C03634=1032.033,-127.655,419.717,167.368,40.722,157.558
C03635=1032.027,-127.904,419.726,167.365,40.724,157.558
C03636=1032.022,-128.154,419.734,167.362,40.725,157.558
C03637=1032.017,-128.403,419.744,167.360,40.726,157.558
C03638=1032.014,-128.653,419.755,167.357,40.726,157.558
C03639=1032.010,-128.903,419.765,167.355,40.727,157.558
C03640=1032.008,-129.153,419.777,167.353,40.725,157.558
C03641=1032.006,-129.403,419.789,167.351,40.724,157.557
C03642=1032.004,-129.653,419.801,167.348,40.723,157.557
C03643=1032.004,-129.903,419.815,167.346,40.721,157.557
C03644=1032.004,-130.152,419.829,167.344,40.719,157.556
C03645=1032.005,-130.402,419.843,167.343,40.715,157.556
C03646=1032.006,-130.653,419.858,167.341,40.712,157.555
C03647=1032.008,-130.902,419.873,167.339,40.709,157.554
C03648=1032.011,-131.152,419.889,167.337,40.704,157.553
C03649=1032.014,-131.402,419.906,167.336,40.699,157.553
C03650=1032.018,-131.653,419.923,167.335,40.694,157.552
C03651=1032.023,-131.902,419.941,167.334,40.688,157.551
C03652=1032.029,-132.152,419.959,167.332,40.682,157.550
C03653=1031.703,-132.177,419.665,167.284,40.914,157.586
C03654=1031.699,-131.927,419.646,167.284,40.920,157.587
C03655=1031.694,-131.678,419.628,167.285,40.927,157.588
C03656=1031.690,-131.428,419.611,167.288,40.932,157.589
C03657=1031.686,-131.177,419.594,167.289,40.937,157.590
C03658=1031.683,-130.928,419.578,167.291,40.941,157.591
C03659=1031.681,-130.677,419.563,167.291,40.945,157.591
C03660=1031.680,-130.428,419.548,167.293,40.948,157.592
C03661=1031.679,-130.177,419.533,167.295,40.951,157.593
C03662=1031.679,-129.927,419.520,167.298,40.953,157.593
C03663=1031.680,-129.678,419.506,167.299,40.955,157.594
C03664=1031.681,-129.428,419.494,167.301,40.957,157.594
C03665=1031.683,-129.178,419.482,167.304,40.958,157.594
C03666=1031.685,-128.928,419.471,167.306,40.959,157.594
C03667=1031.689,-128.678,419.460,167.309,40.959,157.595
C03668=1031.693,-128.428,419.449,167.311,40.959,157.595
C03669=1031.696,-128.179,419.439,167.314,40.958,157.595
C03670=1031.702,-127.929,419.430,167.317,40.956,157.595
C03671=1031.708,-127.679,419.422,167.320,40.954,157.594
C03672=1031.714,-127.430,419.413,167.322,40.953,157.594
C03673=1031.719,-127.181,419.405,167.325,40.951,157.594
C03674=1031.726,-126.931,419.396,167.328,40.949,157.594
C03675=1031.731,-126.681,419.388,167.331,40.948,157.594
C03676=1031.736,-126.431,419.379,167.333,40.946,157.594
C03677=1031.743,-126.182,419.371,167.336,40.944,157.594
C03678=1031.748,-125.932,419.362,167.339,40.942,157.593
C03679=1031.755,-125.682,419.354,167.343,40.941,157.593
C03680=1031.760,-125.432,419.345,167.345,40.939,157.593
C03681=1031.766,-125.182,419.336,167.348,40.937,157.593
C03682=1031.772,-124.933,419.328,167.351,40.936,157.593
C03683=1031.778,-124.683,419.319,167.353,40.934,157.593
C03684=1031.784,-124.433,419.310,167.356,40.932,157.593
C03685=1031.790,-124.183,419.303,167.359,40.931,157.592
C03686=1031.796,-123.934,419.293,167.362,40.929,157.592
C03687=1031.801,-123.684,419.285,167.364,40.927,157.592
C03688=1031.807,-123.434,419.276,167.367,40.925,157.592
C03689=1031.813,-123.184,419.268,167.371,40.924,157.592
C03690=1031.819,-122.934,419.258,167.374,40.922,157.592
C03691=1031.824,-122.685,419.250,167.376,40.920,157.592
C03692=1031.831,-122.434,419.241,167.379,40.919,157.591
C03693=1031.837,-122.185,419.232,167.382,40.917,157.591
C03694=1031.842,-121.935,419.223,167.385,40.915,157.591
C03695=1031.848,-121.686,419.214,167.387,40.913,157.591
C03696=1031.854,-121.435,419.205,167.390,40.912,157.591
C03697=1031.860,-121.186,419.197,167.393,40.910,157.591
C03698=1031.866,-120.936,419.188,167.396,40.908,157.591
C03699=1031.871,-120.687,419.179,167.398,40.907,157.590
C03700=1031.877,-120.436,419.171,167.401,40.905,157.590
C03701=1031.883,-120.187,419.162,167.405,40.903,157.590
C03702=1031.888,-119.973,419.154,167.407,40.902,157.590
C03703=1031.893,-119.760,419.146,167.409,40.901,157.590
C03704=1031.898,-119.546,419.139,167.411,40.899,157.590
C03705=1031.903,-119.332,419.131,167.414,40.898,157.590
C03706=1031.908,-119.118,419.124,167.417,40.896,157.590
C03707=1031.914,-118.904,419.116,167.419,40.895,157.589
C03708=1031.918,-118.690,419.108,167.421,40.894,157.589
C03709=1031.924,-118.477,419.101,167.424,40.892,157.589
C03710=1031.929,-118.226,419.092,167.427,40.890,157.589
C03711=1031.936,-117.977,419.082,167.430,40.889,157.589
C03712=1031.942,-117.727,419.074,167.432,40.887,157.589
C03713=1031.948,-117.477,419.065,167.435,40.885,157.589
C03714=1031.956,-117.119,419.051,167.439,40.884,157.589
C03715=1031.965,-116.761,419.039,167.443,40.881,157.588
C03716=1031.973,-116.403,419.026,167.447,40.878,157.588
C03717=1031.981,-116.044,419.013,167.452,40.877,157.588
C03718=1031.987,-115.794,419.004,167.455,40.875,157.588
C03719=1031.994,-115.544,418.995,167.457,40.873,157.588
C03720=1031.999,-115.295,418.986,167.460,40.872,157.588
C03721=1032.005,-115.045,418.977,167.463,40.870,157.587
C03722=1032.011,-114.795,418.967,167.466,40.868,157.587
C03723=1032.016,-114.545,418.959,167.468,40.867,157.587
C03724=1032.023,-114.295,418.949,167.471,40.865,157.587
C03725=1032.029,-114.045,418.940,167.474,40.864,157.587
C03726=1032.034,-113.796,418.931,167.477,40.862,157.587
C03727=1032.040,-113.546,418.922,167.479,40.860,157.587
C03728=1032.046,-113.296,418.913,167.482,40.859,157.587
C03729=1032.052,-113.047,418.904,167.485,40.858,157.586
C03730=1032.058,-112.797,418.894,167.488,40.856,157.586
C03731=1032.064,-112.547,418.884,167.491,40.854,157.586
C03732=1032.069,-112.297,418.876,167.493,40.853,157.586
C03733=1032.075,-112.047,418.866,167.496,40.852,157.586
C03734=1032.082,-111.798,418.857,167.499,40.850,157.586
C03735=1032.087,-111.549,418.848,167.502,40.848,157.586
C03736=1032.093,-111.298,418.839,167.504,40.847,157.586
C03737=1032.099,-111.048,418.829,167.508,40.846,157.586
C03738=1032.105,-110.799,418.820,167.511,40.844,157.585
C03739=1032.111,-110.549,418.810,167.514,40.842,157.585
C03740=1032.117,-110.299,418.802,167.516,40.840,157.585
C03741=1032.123,-110.049,418.792,167.519,40.839,157.585
C03742=1032.129,-109.799,418.782,167.522,40.838,157.585
C03743=1032.135,-109.550,418.773,167.525,40.836,157.585
C03744=1032.141,-109.301,418.764,167.528,40.834,157.585
C03745=1032.147,-109.051,418.754,167.530,40.833,157.585
C03746=1032.153,-108.800,418.745,167.533,40.832,157.584
C03747=1032.159,-108.551,418.736,167.536,40.830,157.584
C03748=1032.165,-108.301,418.726,167.539,40.828,157.584
C03749=1032.171,-108.052,418.717,167.542,40.827,157.584
C03750=1032.177,-107.802,418.707,167.544,40.826,157.584
C03751=1032.183,-107.552,418.698,167.547,40.824,157.584
C03752=1032.189,-107.302,418.688,167.550,40.822,157.584
C03753=1032.195,-107.053,418.679,167.553,40.821,157.584
C03754=1032.200,-106.803,418.669,167.555,40.820,157.583
C03755=1032.206,-106.553,418.660,167.558,40.818,157.583
C03756=1032.212,-106.303,418.650,167.561,40.817,157.583
C03757=1032.219,-106.053,418.641,167.564,40.815,157.583
C03758=1032.224,-105.804,418.632,167.567,40.814,157.583
C03759=1032.230,-105.554,418.622,167.569,40.813,157.583
C03760=1032.236,-105.304,418.612,167.572,40.811,157.583
C03761=1032.242,-105.054,418.602,167.575,40.810,157.583
C03762=1032.248,-104.804,418.593,167.578,40.808,157.583
C03763=1032.254,-104.555,418.583,167.581,40.807,157.582
C03764=1032.260,-104.306,418.574,167.583,40.806,157.582
C03765=1032.265,-104.055,418.564,167.586,40.804,157.582
C03766=1032.272,-103.806,418.554,167.589,40.803,157.582
C03767=1032.278,-103.556,418.544,167.592,40.801,157.582
C03768=1032.284,-103.307,418.534,167.595,40.800,157.582
C03769=1032.290,-103.057,418.525,167.597,40.799,157.582
C03770=1032.296,-102.807,418.515,167.600,40.797,157.582
C03771=1032.302,-102.557,418.505,167.603,40.796,157.582
C03772=1032.308,-102.307,418.496,167.606,40.794,157.582
C03773=1032.314,-102.058,418.486,167.609,40.793,157.581
C03774=1032.319,-101.808,418.476,167.611,40.792,157.581
C03775=1032.325,-101.558,418.467,167.614,40.790,157.581
C03776=1032.332,-101.309,418.456,167.617,40.789,157.581
C03777=1032.338,-101.059,418.447,167.620,40.787,157.581
C03778=1032.344,-100.772,418.435,167.624,40.785,157.581
C03779=1032.351,-100.485,418.424,167.626,40.784,157.581
C03780=1032.358,-100.198,418.413,167.629,40.783,157.581
C03781=1032.365,-99.911,418.402,167.633,40.781,157.581
C03782=1032.371,-99.661,418.392,167.636,40.779,157.580
C03783=1032.377,-99.412,418.382,167.639,40.778,157.580
C03784=1032.383,-99.162,418.372,167.641,40.777,157.580
C03785=1032.389,-98.912,418.362,167.644,40.775,157.580
C03786=1032.395,-98.662,418.352,167.647,40.774,157.580
C03787=1032.401,-98.413,418.342,167.650,40.772,157.580
C03788=1032.408,-98.163,418.332,167.653,40.771,157.580
C03789=1032.414,-97.913,418.323,167.655,40.770,157.580
C03790=1032.419,-97.663,418.313,167.658,40.768,157.580
C03791=1032.426,-97.414,418.302,167.661,40.767,157.580
C03792=1032.431,-97.164,418.292,167.664,40.766,157.580
C03793=1032.437,-96.914,418.283,167.667,40.764,157.579
C03794=1032.443,-96.665,418.272,167.670,40.763,157.579
C03795=1032.449,-96.415,418.262,167.672,40.762,157.579
C03796=1032.455,-96.165,418.252,167.674,40.761,157.579
C03797=1032.461,-95.916,418.242,167.677,40.760,157.579
C03798=1032.466,-95.665,418.232,167.680,40.758,157.579
C03799=1032.473,-95.416,418.221,167.683,40.757,157.579
C03800=1032.478,-95.166,418.211,167.686,40.756,157.579
C03801=1032.485,-94.916,418.202,167.688,40.754,157.579
C03802=1032.490,-94.667,418.191,167.691,40.753,157.579
C03803=1032.496,-94.417,418.181,167.694,40.752,157.579
C03804=1032.502,-94.168,418.170,167.697,40.751,157.579
C03805=1032.508,-93.918,418.161,167.700,40.750,157.579
C03806=1032.514,-93.668,418.150,167.702,40.748,157.578
C03807=1032.520,-93.417,418.139,167.705,40.747,157.578
C03808=1032.527,-93.168,418.129,167.708,40.746,157.578
C03809=1032.532,-92.918,418.119,167.711,40.744,157.578
C03810=1032.539,-92.669,418.109,167.714,40.743,157.578
C03811=1032.544,-92.419,418.098,167.716,40.742,157.578
C03812=1032.550,-92.170,418.088,167.718,40.741,157.578
C03813=1032.556,-91.920,418.078,167.721,40.740,157.578
C03814=1032.562,-91.670,418.068,167.724,40.738,157.578
C03815=1032.568,-91.420,418.058,167.727,40.737,157.578
C03816=1032.574,-91.171,418.047,167.730,40.736,157.578
C03817=1032.580,-90.921,418.037,167.733,40.734,157.577
C03818=1032.586,-90.671,418.026,167.736,40.733,157.577
C03819=1032.593,-90.422,418.016,167.738,40.732,157.577
C03820=1032.598,-90.172,418.005,167.741,40.731,157.577
C03821=1032.604,-89.922,417.995,167.744,40.730,157.577
C03822=1032.610,-89.672,417.985,167.747,40.728,157.577
C03823=1032.616,-89.423,417.975,167.750,40.727,157.577
C03824=1032.622,-89.174,417.964,167.752,40.726,157.577
C03825=1032.628,-88.923,417.953,167.754,40.725,157.577
C03826=1032.635,-88.674,417.943,167.757,40.724,157.577
C03827=1032.640,-88.423,417.933,167.760,40.723,157.577
C03828=1032.647,-88.174,417.923,167.763,40.721,157.577
C03829=1032.652,-87.925,417.912,167.766,40.720,157.577
C03830=1032.658,-87.674,417.901,167.768,40.718,157.576
C03831=1032.665,-87.425,417.891,167.771,40.717,157.576
C03832=1032.671,-87.175,417.880,167.774,40.716,157.576
C03833=1032.677,-86.926,417.870,167.777,40.715,157.576
C03834=1032.682,-86.676,417.860,167.780,40.714,157.576
C03835=1032.689,-86.426,417.849,167.783,40.713,157.576
C03836=1032.695,-86.177,417.838,167.786,40.711,157.576
C03837=1032.701,-85.927,417.828,167.787,40.710,157.576
C03838=1032.707,-85.677,417.818,167.790,40.709,157.576
C03839=1032.713,-85.427,417.806,167.793,40.707,157.576
C03840=1032.720,-85.178,417.796,167.796,40.706,157.576
C03841=1032.725,-84.928,417.786,167.799,40.705,157.576
C03842=1032.732,-84.643,417.774,167.802,40.704,157.576
C03843=1032.740,-84.359,417.761,167.805,40.703,157.575
C03844=1032.746,-84.074,417.749,167.808,40.701,157.575
C03845=1032.753,-83.789,417.737,167.811,40.699,157.575
C03846=1032.760,-83.539,417.726,167.814,40.698,157.575
C03847=1032.766,-83.289,417.716,167.817,40.697,157.575
C03848=1032.771,-83.040,417.705,167.819,40.696,157.575
C03849=1032.779,-82.790,417.695,167.822,40.695,157.575
C03850=1032.784,-82.540,417.684,167.825,40.694,157.575
C03851=1032.790,-82.291,417.673,167.828,40.692,157.575
C03852=1032.797,-82.041,417.662,167.831,40.691,157.575
C03853=1032.803,-81.792,417.651,167.834,40.690,157.575
C03854=1032.809,-81.542,417.642,167.837,40.688,157.575
C03855=1032.815,-81.292,417.631,167.839,40.687,157.574
C03856=1032.821,-81.042,417.620,167.841,40.687,157.574
C03857=1032.828,-80.793,417.609,167.844,40.685,157.574
C03858=1032.834,-80.543,417.598,167.847,40.684,157.574
C03859=1032.840,-80.293,417.587,167.850,40.683,157.574
C03860=1032.846,-80.044,417.577,167.853,40.681,157.574
C03861=1032.852,-79.794,417.566,167.855,40.680,157.574
C03862=1032.858,-79.544,417.555,167.858,40.679,157.574
C03863=1032.864,-79.295,417.544,167.861,40.678,157.574
C03864=1032.870,-79.045,417.533,167.863,40.677,157.574
C03865=1032.876,-78.795,417.522,167.866,40.676,157.574
C03866=1032.883,-78.545,417.511,167.869,40.675,157.574
C03867=1032.889,-78.296,417.500,167.872,40.674,157.574
C03868=1032.895,-78.046,417.490,167.875,40.673,157.574
C03869=1032.901,-77.796,417.478,167.877,40.672,157.574
C03870=1032.907,-77.547,417.467,167.880,40.671,157.574
C03871=1032.912,-77.297,417.457,167.882,40.670,157.573
C03872=1032.919,-77.047,417.445,167.885,40.668,157.573
C03873=1032.924,-76.797,417.434,167.888,40.667,157.573
C03874=1032.932,-76.548,417.423,167.891,40.666,157.573
C03875=1032.938,-76.299,417.412,167.894,40.665,157.573
C03876=1032.943,-76.049,417.401,167.896,40.664,157.573
C03877=1032.950,-75.799,417.390,167.899,40.663,157.573
C03878=1032.955,-75.550,417.379,167.901,40.662,157.573
C03879=1032.962,-75.299,417.368,167.904,40.661,157.573
C03880=1032.968,-75.050,417.357,167.907,40.660,157.573
C03881=1032.974,-74.800,417.345,167.910,40.659,157.573
C03882=1032.980,-74.551,417.334,167.913,40.658,157.573
C03883=1032.986,-74.301,417.323,167.916,40.657,157.573
C03884=1032.992,-74.051,417.312,167.917,40.656,157.573
C03885=1032.998,-73.801,417.301,167.920,40.655,157.573
C03886=1033.004,-73.552,417.289,167.923,40.654,157.573
C03887=1033.010,-73.303,417.278,167.926,40.653,157.573
C03888=1033.016,-73.052,417.267,167.929,40.652,157.573
C03889=1033.022,-72.803,417.256,167.931,40.651,157.573
C03890=1033.028,-72.553,417.244,167.934,40.650,157.572
C03891=1033.034,-72.303,417.233,167.937,40.649,157.572
C03892=1033.040,-72.054,417.221,167.940,40.648,157.572
C03893=1033.046,-71.804,417.210,167.941,40.647,157.572
C03894=1033.053,-71.554,417.199,167.944,40.646,157.572
C03895=1033.058,-71.305,417.187,167.947,40.645,157.572
C03896=1033.064,-71.055,417.175,167.950,40.644,157.572
C03897=1033.070,-70.805,417.164,167.953,40.643,157.572
C03898=1033.077,-70.556,417.152,167.955,40.642,157.572
C03899=1033.082,-70.306,417.142,167.958,40.642,157.572
C03900=1033.088,-70.056,417.129,167.961,40.641,157.572
C03901=1033.094,-69.807,417.118,167.964,40.640,157.572
C03902=1033.100,-69.557,417.107,167.966,40.639,157.572
C03903=1033.106,-69.308,417.095,167.968,40.638,157.572
C03904=1033.113,-69.058,417.084,167.971,40.637,157.572
C03905=1033.118,-68.808,417.072,167.974,40.636,157.572
C03906=1033.125,-68.526,417.059,167.977,40.635,157.572
C03907=1033.132,-68.243,417.046,167.980,40.634,157.572
C03908=1033.139,-67.961,417.033,167.983,40.633,157.572
C03909=1033.146,-67.677,417.020,167.986,40.632,157.572
C03910=1033.151,-67.428,417.009,167.989,40.631,157.572
C03911=1033.158,-67.178,416.997,167.992,40.630,157.572
C03912=1033.164,-66.929,416.986,167.994,40.629,157.572
C03913=1033.170,-66.679,416.974,167.996,40.629,157.572
C03914=1033.176,-66.429,416.963,167.999,40.628,157.572
C03915=1033.182,-66.180,416.950,168.002,40.627,157.572
C03916=1033.189,-65.930,416.938,168.005,40.626,157.572
C03917=1033.194,-65.681,416.928,168.007,40.625,157.571
C03918=1033.201,-65.431,416.916,168.010,40.624,157.571
C03919=1033.206,-65.181,416.904,168.013,40.623,157.571
C03920=1033.213,-64.932,416.892,168.016,40.622,157.571
C03921=1033.219,-64.681,416.881,168.017,40.621,157.571
C03922=1033.225,-64.433,416.869,168.020,40.620,157.571
C03923=1033.231,-64.183,416.857,168.023,40.619,157.571
C03924=1033.237,-63.932,416.846,168.026,40.618,157.571
C03925=1033.243,-63.684,416.834,168.028,40.617,157.571
C03926=1033.250,-63.433,416.823,168.031,40.616,157.571
C03927=1033.256,-63.184,416.811,168.034,40.615,157.571
C03928=1033.262,-62.935,416.799,168.037,40.615,157.571
C03929=1033.268,-62.684,416.787,168.040,40.614,157.571
C03930=1033.275,-62.435,416.775,168.042,40.613,157.571
C03931=1033.281,-62.186,416.764,168.044,40.612,157.571
C03932=1033.286,-61.935,416.752,168.047,40.611,157.571
C03933=1033.293,-61.686,416.740,168.050,40.610,157.571
C03934=1033.299,-61.437,416.728,168.052,40.609,157.571
C03935=1033.305,-61.187,416.717,168.055,40.608,157.571
C03936=1033.311,-60.937,416.705,168.058,40.607,157.571
C03937=1033.318,-60.687,416.693,168.061,40.606,157.571
C03938=1033.324,-60.438,416.682,168.063,40.605,157.571
C03939=1033.330,-60.188,416.669,168.066,40.604,157.571
C03940=1033.336,-59.938,416.657,168.068,40.603,157.571
C03941=1033.343,-59.689,416.645,168.071,40.602,157.571
C03942=1033.349,-59.439,416.634,168.073,40.602,157.570
C03943=1033.354,-59.190,416.622,168.076,40.601,157.570
C03944=1033.361,-58.940,416.610,168.079,40.600,157.570
C03945=1033.368,-58.690,416.598,168.082,40.599,157.571
C03946=1033.373,-58.441,416.586,168.084,40.598,157.570
C03947=1033.379,-58.191,416.575,168.087,40.597,157.570
C03948=1033.386,-57.941,416.563,168.090,40.596,157.570
C03949=1033.393,-57.692,416.551,168.092,40.596,157.570
C03950=1033.399,-57.442,416.538,168.094,40.595,157.570
C03951=1033.405,-57.193,416.526,168.097,40.594,157.570
C03952=1033.411,-56.943,416.515,168.100,40.593,157.570
C03953=1033.417,-56.693,416.503,168.102,40.592,157.570
C03954=1033.424,-56.443,416.491,168.105,40.591,157.570
C03955=1033.430,-56.194,416.479,168.108,40.590,157.570
C03956=1033.436,-55.945,416.467,168.111,40.589,157.570
C03957=1033.442,-55.695,416.455,168.113,40.588,157.570
C03958=1033.449,-55.446,416.443,168.116,40.587,157.570
C03959=1033.455,-55.195,416.431,168.118,40.586,157.570
C03960=1033.461,-54.945,416.419,168.121,40.585,157.570
C03961=1033.468,-54.696,416.407,168.123,40.585,157.570
C03962=1033.474,-54.446,416.395,168.126,40.584,157.570
C03963=1033.480,-54.197,416.383,168.129,40.583,157.570
C03964=1033.486,-53.948,416.371,168.132,40.582,157.570
C03965=1033.493,-53.698,416.359,168.134,40.581,157.570
C03966=1033.499,-53.448,416.346,168.137,40.580,157.570
C03967=1033.505,-53.199,416.334,168.140,40.579,157.570
C03968=1033.512,-52.949,416.322,168.142,40.578,157.570
C03969=1033.519,-52.699,416.310,168.144,40.577,157.570
C03970=1033.525,-52.418,416.297,168.147,40.576,157.569
C03971=1033.533,-52.137,416.283,168.150,40.575,157.569
C03972=1033.540,-51.855,416.269,168.153,40.574,157.569
C03973=1033.547,-51.574,416.256,168.156,40.573,157.569
C03974=1033.553,-51.324,416.243,168.159,40.572,157.569
C03975=1033.560,-51.075,416.231,168.162,40.571,157.569
C03976=1033.566,-50.825,416.219,168.165,40.570,157.569
C03977=1033.572,-50.575,416.206,168.167,40.569,157.569
C03978=1033.579,-50.326,416.194,168.169,40.568,157.569
C03979=1033.585,-50.076,416.182,168.173,40.568,157.569
C03980=1033.591,-49.826,416.169,168.174,40.567,157.569
C03981=1033.597,-49.576,416.157,168.177,40.566,157.569
C03982=1033.603,-49.327,416.145,168.180,40.566,157.569
C03983=1033.609,-49.078,416.132,168.182,40.565,157.569
C03984=1033.616,-48.828,416.120,168.185,40.564,157.569
C03985=1033.621,-48.578,416.107,168.187,40.563,157.569
C03986=1033.627,-48.329,416.095,168.190,40.563,157.569
C03987=1033.634,-48.079,416.083,168.193,40.562,157.569
C03988=1033.640,-47.830,416.070,168.195,40.561,157.569
C03989=1033.646,-47.580,416.057,168.198,40.561,157.569
C03990=1033.652,-47.330,416.045,168.201,40.560,157.569
C03991=1033.659,-47.080,416.033,168.203,40.559,157.569
C03992=1033.665,-46.831,416.019,168.206,40.559,157.569
C03993=1033.671,-46.581,416.007,168.209,40.558,157.569
C03994=1033.677,-46.332,415.995,168.210,40.557,157.569
C03995=1033.683,-46.082,415.982,168.213,40.556,157.569
C03996=1033.690,-45.833,415.969,168.215,40.556,157.569
C03997=1033.696,-45.583,415.957,168.218,40.555,157.569
C03998=1033.702,-45.333,415.944,168.221,40.554,157.569
C03999=1033.708,-45.084,415.931,168.223,40.553,157.569
C04000=1033.714,-44.834,415.919,168.226,40.552,157.569
C04001=1033.721,-44.584,415.907,168.229,40.551,157.569
C04002=1033.727,-44.335,415.893,168.231,40.551,157.569
C04003=1033.733,-44.085,415.881,168.234,40.550,157.569
C04004=1033.740,-43.836,415.869,168.236,40.549,157.569
C04005=1033.746,-43.586,415.856,168.239,40.549,157.569
C04006=1033.752,-43.337,415.843,168.242,40.548,157.569
C04007=1033.758,-43.087,415.830,168.244,40.547,157.569
C04008=1033.765,-42.838,415.818,168.246,40.546,157.569
C04009=1033.771,-42.588,415.805,168.249,40.546,157.569
C04010=1033.777,-42.339,415.792,168.251,40.545,157.569
C04011=1033.783,-42.089,415.779,168.254,40.544,157.569
C04012=1033.790,-41.840,415.767,168.256,40.544,157.569
C04013=1033.796,-41.590,415.754,168.259,40.543,157.569
C04014=1033.802,-41.339,415.741,168.262,40.542,157.569
C04015=1033.808,-41.090,415.728,168.264,40.542,157.569
C04016=1033.815,-40.840,415.716,168.267,40.541,157.569
C04017=1033.821,-40.591,415.703,168.270,40.540,157.569
C04018=1033.827,-40.341,415.690,168.272,40.539,157.569
C04019=1033.833,-40.092,415.677,168.275,40.539,157.569
C04020=1033.840,-39.842,415.665,168.277,40.538,157.569
C04021=1033.846,-39.593,415.652,168.279,40.537,157.569
C04022=1033.852,-39.343,415.639,168.283,40.536,157.569
C04023=1033.859,-39.093,415.626,168.284,40.536,157.569
C04024=1033.865,-38.844,415.614,168.287,40.535,157.569
C04025=1033.872,-38.594,415.600,168.289,40.534,157.569
C04026=1033.878,-38.345,415.588,168.292,40.533,157.569
C04027=1033.884,-38.095,415.574,168.295,40.533,157.569
C04028=1033.890,-37.846,415.561,168.297,40.532,157.569
C04029=1033.896,-37.596,415.549,168.300,40.531,157.569
C04030=1033.903,-37.346,415.535,168.302,40.531,157.569
C04031=1033.909,-37.097,415.522,168.305,40.530,157.569
C04032=1033.915,-36.847,415.509,168.307,40.530,157.569
C04033=1033.921,-36.598,415.496,168.310,40.529,157.569
C04034=1033.928,-36.316,415.481,168.313,40.529,157.569
C04035=1033.935,-36.036,415.466,168.316,40.528,157.569
C04036=1033.942,-35.755,415.452,168.319,40.527,157.569
C04037=1033.948,-35.474,415.437,168.321,40.526,157.569
C04038=1033.954,-35.224,415.424,168.324,40.526,157.569
C04039=1033.961,-34.974,415.410,168.327,40.525,157.569
C04040=1033.967,-34.724,415.398,168.328,40.524,157.569
C04041=1033.973,-34.475,415.384,168.332,40.524,157.569
C04042=1033.979,-34.226,415.371,168.333,40.523,157.569
C04043=1033.986,-33.977,415.358,168.336,40.522,157.569
C04044=1033.992,-33.726,415.345,168.338,40.522,157.569
C04045=1033.998,-33.477,415.332,168.341,40.521,157.569
C04046=1034.005,-33.228,415.318,168.343,40.521,157.569
C04047=1034.011,-32.978,415.305,168.346,40.520,157.569
C04048=1034.017,-32.728,415.292,168.348,40.520,157.569
C04049=1034.024,-32.478,415.279,168.351,40.519,157.569
C04050=1034.030,-32.229,415.266,168.354,40.518,157.569
C04051=1034.036,-31.980,415.252,168.356,40.517,157.569
C04052=1034.043,-31.730,415.239,168.359,40.516,157.569
C04053=1034.049,-31.480,415.226,168.361,40.516,157.569
C04054=1034.055,-31.231,415.213,168.364,40.515,157.569
C04055=1034.061,-30.982,415.200,168.366,40.515,157.569
C04056=1034.068,-30.732,415.186,168.369,40.514,157.569
C04057=1034.074,-30.482,415.173,168.371,40.514,157.569
C04058=1034.080,-30.233,415.159,168.374,40.513,157.569
C04059=1034.087,-29.984,415.146,168.375,40.512,157.569
C04060=1034.093,-29.733,415.133,168.379,40.512,157.569
C04061=1034.099,-29.484,415.120,168.380,40.511,157.569
C04062=1034.106,-29.235,415.107,168.383,40.511,157.569
C04063=1034.112,-28.985,415.093,168.386,40.510,157.569
C04064=1034.119,-28.735,415.080,168.388,40.509,157.569
C04065=1034.125,-28.486,415.067,168.391,40.508,157.569
C04066=1034.131,-28.236,415.052,168.393,40.508,157.569
C04067=1034.137,-27.987,415.039,168.396,40.507,157.569
C04068=1034.143,-27.737,415.026,168.398,40.506,157.569
C04069=1034.150,-27.487,415.012,168.401,40.506,157.569
C04070=1034.156,-27.238,414.999,168.403,40.505,157.569
C04071=1034.163,-26.989,414.986,168.406,40.505,157.569
C04072=1034.169,-26.739,414.972,168.408,40.504,157.569
C04073=1034.175,-26.489,414.958,168.411,40.504,157.569
C04074=1034.181,-26.240,414.945,168.413,40.503,157.569
C04075=1034.188,-25.990,414.931,168.416,40.503,157.569
C04076=1034.193,-25.741,414.917,168.418,40.502,157.569
C04077=1034.200,-25.491,414.904,168.421,40.501,157.569
C04078=1034.206,-25.241,414.890,168.423,40.501,157.569
C04079=1034.213,-24.992,414.877,168.426,40.500,157.569
C04080=1034.218,-24.742,414.863,168.428,40.500,157.569
C04081=1034.225,-24.492,414.850,168.431,40.499,157.569
C04082=1034.231,-24.243,414.836,168.433,40.499,157.569
C04083=1034.237,-23.993,414.822,168.435,40.499,157.569
C04084=1034.243,-23.744,414.809,168.437,40.498,157.569
C04085=1034.250,-23.495,414.795,168.440,40.497,157.569
C04086=1034.256,-23.245,414.781,168.442,40.497,157.569
C04087=1034.262,-22.995,414.767,168.444,40.496,157.569
C04088=1034.268,-22.746,414.754,168.447,40.496,157.569
C04089=1034.274,-22.496,414.740,168.449,40.495,157.569
C04090=1034.281,-22.247,414.727,168.452,40.495,157.569
C04091=1034.288,-21.997,414.712,168.454,40.494,157.569
C04092=1034.293,-21.748,414.698,168.457,40.494,157.569
C04093=1034.300,-21.499,414.685,168.459,40.493,157.569
C04094=1034.306,-21.249,414.671,168.462,40.492,157.569
C04095=1034.312,-20.999,414.658,168.464,40.492,157.569
C04096=1034.319,-20.750,414.643,168.467,40.491,157.569
C04097=1034.325,-20.500,414.630,168.469,40.491,157.569
C04098=1034.332,-20.218,414.615,168.472,40.490,157.569
C04099=1034.339,-19.937,414.599,168.475,40.490,157.569
C04100=1034.347,-19.654,414.583,168.477,40.489,157.569
C04101=1034.353,-19.373,414.568,168.480,40.489,157.569
C04102=1034.360,-19.123,414.554,168.483,40.488,157.569
C04103=1034.366,-18.874,414.540,168.485,40.487,157.569
C04104=1034.373,-18.624,414.526,168.487,40.487,157.569
C04105=1034.378,-18.375,414.512,168.490,40.486,157.569
C04106=1034.385,-18.125,414.498,168.492,40.485,157.569
C04107=1034.392,-17.876,414.484,168.495,40.485,157.569
C04108=1034.398,-17.626,414.470,168.497,40.485,157.569
C04109=1034.404,-17.377,414.457,168.500,40.484,157.569
C04110=1034.411,-17.127,414.443,168.502,40.484,157.569
C04111=1034.417,-16.878,414.429,168.505,40.483,157.569
C04112=1034.423,-16.628,414.415,168.507,40.483,157.569
C04113=1034.429,-16.379,414.400,168.509,40.482,157.569
C04114=1034.436,-16.129,414.387,168.511,40.481,157.569
C04115=1034.442,-15.880,414.373,168.513,40.481,157.569
C04116=1034.449,-15.630,414.359,168.516,40.480,157.569
C04117=1034.455,-15.380,414.345,168.518,40.479,157.569
C04118=1034.461,-15.131,414.330,168.521,40.479,157.569
C04119=1034.468,-14.881,414.317,168.523,40.479,157.569
C04120=1034.474,-14.632,414.302,168.525,40.479,157.569
C04121=1034.481,-14.382,414.289,168.528,40.478,157.569
C04122=1034.486,-14.133,414.274,168.530,40.477,157.569
C04123=1034.492,-13.883,414.260,168.533,40.477,157.569
C04124=1034.499,-13.634,414.246,168.535,40.476,157.569
C04125=1034.505,-13.384,414.232,168.537,40.476,157.569
C04126=1034.511,-13.135,414.217,168.540,40.476,157.569
C04127=1034.518,-12.885,414.203,168.542,40.475,157.569
C04128=1034.523,-12.636,414.189,168.545,40.475,157.570
C04129=1034.530,-12.386,414.175,168.547,40.474,157.570
C04130=1034.537,-12.136,414.160,168.549,40.474,157.569
C04131=1034.542,-11.887,414.146,168.552,40.473,157.570
C04132=1034.549,-11.638,414.132,168.554,40.473,157.570
C04133=1034.555,-11.389,414.117,168.557,40.473,157.570
C04134=1034.562,-11.139,414.104,168.559,40.472,157.570
C04135=1034.568,-10.890,414.089,168.561,40.472,157.570
C04136=1034.574,-10.639,414.075,168.564,40.471,157.570
C04137=1034.581,-10.390,414.061,168.566,40.470,157.570
C04138=1034.587,-10.141,414.046,168.569,40.470,157.570
C04139=1034.593,-9.891,414.032,168.571,40.470,157.570
C04140=1034.600,-9.641,414.017,168.573,40.469,157.570
C04141=1034.605,-9.392,414.004,168.576,40.469,157.570
C04142=1034.612,-9.142,413.989,168.578,40.469,157.570
C04143=1034.618,-8.894,413.975,168.580,40.468,157.570
C04144=1034.624,-8.643,413.960,168.583,40.467,157.570
C04145=1034.631,-8.394,413.945,168.585,40.467,157.570
C04146=1034.637,-8.145,413.931,168.588,40.466,157.570
C04147=1034.643,-7.895,413.917,168.590,40.466,157.570
C04148=1034.650,-7.645,413.903,168.592,40.466,157.570
C04149=1034.656,-7.396,413.888,168.595,40.465,157.570
C04150=1034.662,-7.146,413.874,168.597,40.465,157.570
C04151=1034.669,-6.897,413.860,168.599,40.464,157.570
C04152=1034.675,-6.648,413.845,168.602,40.464,157.570
C04153=1034.681,-6.398,413.830,168.604,40.463,157.570
C04154=1034.688,-6.148,413.817,168.607,40.463,157.570
C04155=1034.695,-5.899,413.802,168.609,40.462,157.570
C04156=1034.700,-5.650,413.787,168.611,40.462,157.570
C04157=1034.708,-5.400,413.773,168.614,40.461,157.570
C04158=1034.714,-5.150,413.758,168.616,40.461,157.570
C04159=1034.719,-4.901,413.744,168.618,40.461,157.570
C04160=1034.727,-4.652,413.729,168.620,40.460,157.570
C04161=1034.733,-4.402,413.715,168.622,40.459,157.570
C04162=1034.740,-4.119,413.698,168.626,40.459,157.570
C04163=1034.747,-3.835,413.682,168.628,40.458,157.570
C04164=1034.754,-3.552,413.665,168.630,40.458,157.570
C04165=1034.762,-3.269,413.648,168.633,40.458,157.570
C04166=1034.768,-3.019,413.633,168.635,40.457,157.570
C04167=1034.774,-2.769,413.619,168.639,40.457,157.571
C04168=1034.780,-2.520,413.605,168.640,40.456,157.570
C04169=1034.786,-2.270,413.590,168.642,40.456,157.571
C04170=1034.793,-2.021,413.575,168.644,40.456,157.571
C04171=1034.798,-1.772,413.560,168.647,40.456,157.571
C04172=1034.805,-1.522,413.545,168.650,40.455,157.571
C04173=1034.811,-1.272,413.530,168.652,40.455,157.571
C04174=1034.817,-1.023,413.515,168.654,40.454,157.571
C04175=1034.823,-0.774,413.501,168.656,40.454,157.571
C04176=1034.830,-0.524,413.486,168.658,40.454,157.571
C04177=1034.836,-0.274,413.471,168.662,40.453,157.571
C04178=1034.842,-0.025,413.456,168.664,40.453,157.571
C04179=1034.848,0.224,413.441,168.666,40.453,157.571
C04180=1034.855,0.474,413.426,168.667,40.452,157.571
C04181=1034.861,0.724,413.411,168.670,40.452,157.571
C04182=1034.867,0.973,413.397,168.672,40.452,157.571
C04183=1034.873,1.222,413.382,168.675,40.451,157.571
C04184=1034.880,1.472,413.367,168.678,40.451,157.571
C04185=1034.886,1.722,413.352,168.680,40.451,157.571
C04186=1034.892,1.971,413.337,168.681,40.450,157.571
C04187=1034.899,2.220,413.321,168.684,40.450,157.571
C04188=1034.905,2.469,413.307,168.687,40.450,157.571
C04189=1034.911,2.719,413.292,168.689,40.449,157.571
C04190=1034.918,2.968,413.277,168.691,40.449,157.571
C04191=1034.924,3.218,413.262,168.693,40.448,157.571
C04192=1034.930,3.468,413.247,168.695,40.448,157.571
C04193=1034.936,3.717,413.232,168.697,40.448,157.571
C04194=1034.942,3.966,413.218,168.701,40.447,157.572
C04195=1034.948,4.216,413.202,168.703,40.447,157.572
C04196=1034.955,4.465,413.186,168.704,40.446,157.572
C04197=1034.961,4.715,413.171,168.706,40.446,157.572
C04198=1034.968,4.965,413.156,168.709,40.446,157.572
C04199=1034.973,5.214,413.142,168.712,40.446,157.572
C04200=1034.980,5.463,413.127,168.714,40.446,157.572
C04201=1034.986,5.713,413.112,168.716,40.445,157.572
C04202=1034.993,5.962,413.096,168.718,40.444,157.572
C04203=1034.999,6.212,413.081,168.720,40.444,157.572
C04204=1035.006,6.461,413.066,168.723,40.444,157.572
C04205=1035.012,6.711,413.051,168.726,40.444,157.572
C04206=1035.018,6.961,413.037,168.727,40.443,157.572
C04207=1035.025,7.210,413.021,168.729,40.443,157.572
C04208=1035.031,7.459,413.006,168.732,40.442,157.572
C04209=1035.037,7.708,412.991,168.734,40.442,157.572
C04210=1035.044,7.958,412.976,168.736,40.441,157.572
C04211=1035.050,8.207,412.961,168.738,40.441,157.572
C04212=1035.057,8.457,412.946,168.741,40.441,157.572
C04213=1035.063,8.706,412.931,168.743,40.440,157.572
C04214=1035.069,8.956,412.916,168.745,40.440,157.572
C04215=1035.076,9.205,412.900,168.748,40.439,157.572
C04216=1035.082,9.455,412.885,168.750,40.439,157.572
C04217=1035.088,9.705,412.870,168.752,40.439,157.572
C04218=1035.094,9.954,412.855,168.754,40.439,157.572
C04219=1035.101,10.203,412.839,168.757,40.438,157.572
C04220=1035.108,10.453,412.824,168.759,40.438,157.572
C04221=1035.114,10.703,412.809,168.761,40.437,157.572
C04222=1035.121,10.952,412.794,168.764,40.437,157.573
C04223=1035.127,11.201,412.779,168.766,40.436,157.572
C04224=1035.133,11.451,412.764,168.768,40.436,157.572
C04225=1035.140,11.700,412.748,168.770,40.436,157.573
C04226=1035.147,11.985,412.731,168.773,40.435,157.573
C04227=1035.154,12.270,412.714,168.776,40.434,157.573
C04228=1035.162,12.556,412.696,168.778,40.434,157.573
C04229=1035.169,12.841,412.678,168.781,40.434,157.573
C04230=1035.176,13.090,412.663,168.783,40.434,157.573
C04231=1035.182,13.339,412.648,168.785,40.433,157.573
C04232=1035.189,13.589,412.633,168.788,40.433,157.573
C04233=1035.194,13.839,412.617,168.790,40.432,157.573
C04234=1035.201,14.088,412.602,168.792,40.432,157.573
C04235=1035.208,14.338,412.587,168.794,40.431,157.573
C04236=1035.213,14.587,412.570,168.797,40.431,157.573
C04237=1035.220,14.837,412.555,168.799,40.431,157.573
C04238=1035.227,15.086,412.540,168.801,40.431,157.573
C04239=1035.232,15.336,412.524,168.803,40.430,157.573
C04240=1035.239,15.585,412.509,168.806,40.430,157.573
C04241=1035.245,15.835,412.494,168.808,40.430,157.573
C04242=1035.251,16.084,412.477,168.810,40.430,157.573
C04243=1035.258,16.333,412.462,168.812,40.430,157.573
C04244=1035.264,16.583,412.447,168.814,40.429,157.573
C04245=1035.270,16.832,412.431,168.817,40.428,157.573
C04246=1035.277,17.082,412.416,168.819,40.428,157.573
C04247=1035.283,17.331,412.400,168.821,40.428,157.573
C04248=1035.289,17.581,412.384,168.823,40.428,157.573
C04249=1035.296,17.830,412.368,168.826,40.427,157.574
C04250=1035.303,18.079,412.353,168.828,40.427,157.574
C04251=1035.309,18.329,412.337,168.830,40.427,157.574
C04252=1035.315,18.578,412.322,168.832,40.426,157.574
C04253=1035.322,18.827,412.306,168.834,40.426,157.574
C04254=1035.328,19.077,412.290,168.837,40.426,157.574
C04255=1035.334,19.326,412.275,168.839,40.425,157.574
C04256=1035.341,19.576,412.260,168.841,40.425,157.574
C04257=1035.347,19.825,412.243,168.843,40.425,157.574
C04258=1035.353,20.074,412.228,168.845,40.425,157.574
C04259=1035.359,20.324,412.212,168.849,40.425,157.574
C04260=1035.366,20.573,412.197,168.851,40.424,157.574
C04261=1035.372,20.823,412.180,168.852,40.423,157.574
C04262=1035.379,21.073,412.164,168.854,40.423,157.574
C04263=1035.385,21.323,412.149,168.856,40.423,157.574
C04264=1035.391,21.572,412.133,168.859,40.423,157.574
C04265=1035.397,21.821,412.117,168.862,40.423,157.574
C04266=1035.404,22.070,412.101,168.864,40.422,157.574
C04267=1035.410,22.319,412.085,168.866,40.422,157.574
C04268=1035.416,22.569,412.070,168.868,40.422,157.574
C04269=1035.422,22.818,412.054,168.871,40.422,157.574
C04270=1035.429,23.067,412.038,168.873,40.421,157.574
C04271=1035.435,23.317,412.021,168.875,40.421,157.575
C04272=1035.442,23.567,412.006,168.877,40.421,157.575
C04273=1035.448,23.816,411.990,168.879,40.421,157.575
C04274=1035.454,24.065,411.975,168.882,40.420,157.575
C04275=1035.460,24.315,411.958,168.884,40.420,157.575
C04276=1035.467,24.564,411.943,168.886,40.419,157.575
C04277=1035.473,24.813,411.926,168.888,40.419,157.575
C04278=1035.480,25.064,411.911,168.890,40.419,157.575
C04279=1035.486,25.313,411.895,168.893,40.419,157.575
C04280=1035.492,25.562,411.879,168.895,40.419,157.575
C04281=1035.499,25.811,411.863,168.897,40.418,157.575
C04282=1035.505,26.061,411.847,168.899,40.418,157.575
C04283=1035.512,26.310,411.831,168.901,40.418,157.575
C04284=1035.518,26.560,411.814,168.904,40.417,157.575
C04285=1035.524,26.809,411.799,168.906,40.417,157.575
C04286=1035.530,27.058,411.782,168.908,40.417,157.575
C04287=1035.537,27.308,411.768,168.910,40.416,157.575
C04288=1035.543,27.558,411.751,168.912,40.416,157.575
C04289=1035.549,27.807,411.735,168.914,40.416,157.575
C04290=1035.557,28.093,411.716,168.917,40.416,157.575
C04291=1035.564,28.380,411.697,168.919,40.415,157.575
C04292=1035.571,28.666,411.679,168.922,40.415,157.575
C04293=1035.579,28.953,411.661,168.924,40.415,157.576
C04294=1035.585,29.202,411.645,168.927,40.415,157.576
C04295=1035.590,29.451,411.628,168.929,40.414,157.576
C04296=1035.598,29.701,411.612,168.931,40.414,157.576
C04297=1035.604,29.951,411.596,168.933,40.414,157.576
C04298=1035.610,30.200,411.580,168.935,40.414,157.576
C04299=1035.616,30.449,411.563,168.937,40.414,157.576
C04300=1035.623,30.699,411.547,168.939,40.413,157.576
C04301=1035.629,30.948,411.531,168.942,40.413,157.576
C04302=1035.635,31.197,411.514,168.944,40.413,157.576
C04303=1035.641,31.446,411.498,168.946,40.413,157.576
C04304=1035.648,31.696,411.482,168.948,40.413,157.576
C04305=1035.654,31.945,411.466,168.950,40.412,157.576
C04306=1035.660,32.195,411.449,168.952,40.412,157.576
C04307=1035.666,32.444,411.433,168.955,40.412,157.576
C04308=1035.673,32.694,411.417,168.957,40.412,157.576
C04309=1035.679,32.943,411.401,168.959,40.411,157.576
C04310=1035.685,33.193,411.385,168.961,40.411,157.577
C04311=1035.692,33.441,411.368,168.963,40.411,157.577
C04312=1035.698,33.691,411.351,168.965,40.411,157.577
C04313=1035.705,33.940,411.335,168.967,40.410,157.577
C04314=1035.711,34.190,411.319,168.970,40.410,157.577
C04315=1035.717,34.440,411.302,168.972,40.409,157.577
C04316=1035.723,34.689,411.286,168.974,40.409,157.577
C04317=1035.730,34.938,411.270,168.976,40.409,157.577
C04318=1035.737,35.188,411.253,168.978,40.409,157.577
C04319=1035.743,35.437,411.237,168.980,40.409,157.577
C04320=1035.749,35.686,411.221,168.982,40.408,157.577
C04321=1035.755,35.936,411.204,168.985,40.408,157.577
C04322=1035.762,36.185,411.188,168.988,40.408,157.577
C04323=1035.768,36.434,411.171,168.990,40.408,157.577
C04324=1035.775,36.684,411.155,168.992,40.407,157.577
C04325=1035.781,36.934,411.139,168.994,40.407,157.577
C04326=1035.787,37.182,411.122,168.996,40.407,157.577
C04327=1035.794,37.432,411.106,168.999,40.407,157.577
C04328=1035.800,37.681,411.089,169.001,40.407,157.577
C04329=1035.807,37.930,411.072,169.003,40.406,157.577
C04330=1035.813,38.180,411.056,169.005,40.406,157.578
C04331=1035.819,38.429,411.039,169.007,40.406,157.578
C04332=1035.825,38.678,411.023,169.009,40.406,157.578
C04333=1035.832,38.928,411.006,169.011,40.406,157.578
C04334=1035.838,39.178,410.990,169.013,40.405,157.578
C04335=1035.844,39.426,410.973,169.015,40.405,157.578
C04336=1035.851,39.676,410.956,169.018,40.405,157.578
C04337=1035.857,39.926,410.940,169.020,40.405,157.578
C04338=1035.862,40.175,410.922,169.022,40.404,157.578
C04339=1035.869,40.425,410.906,169.024,40.404,157.578
C04340=1035.875,40.674,410.889,169.026,40.404,157.578
C04341=1035.881,40.924,410.872,169.028,40.404,157.578
C04342=1035.888,41.172,410.855,169.030,40.404,157.578
C04343=1035.894,41.422,410.839,169.032,40.404,157.578
C04344=1035.900,41.672,410.822,169.035,40.404,157.578
C04345=1035.906,41.920,410.805,169.037,40.404,157.578
C04346=1035.912,42.170,410.789,169.039,40.403,157.579
C04347=1035.919,42.419,410.772,169.041,40.403,157.579
C04348=1035.925,42.669,410.755,169.043,40.403,157.579
C04349=1035.932,42.918,410.738,169.045,40.403,157.579
C04350=1035.938,43.167,410.722,169.047,40.403,157.579
C04351=1035.945,43.417,410.704,169.049,40.402,157.579
C04352=1035.951,43.666,410.688,169.051,40.402,157.579
C04353=1035.956,43.915,410.671,169.053,40.402,157.579
C04354=1035.964,44.202,410.652,169.057,40.402,157.579
C04355=1035.971,44.488,410.632,169.059,40.402,157.579
C04356=1035.978,44.775,410.612,169.062,40.402,157.579
C04357=1035.985,45.061,410.593,169.064,40.402,157.579
C04358=1035.991,45.311,410.576,169.066,40.401,157.579
C04359=1035.998,45.559,410.559,169.068,40.401,157.579
C04360=1036.004,45.810,410.542,169.070,40.402,157.580
C04361=1036.010,46.058,410.525,169.072,40.401,157.580
C04362=1036.016,46.308,410.508,169.074,40.401,157.580
C04363=1036.022,46.558,410.490,169.076,40.401,157.580
C04364=1036.028,46.806,410.473,169.078,40.401,157.580
C04365=1036.035,47.056,410.457,169.081,40.400,157.580
C04366=1036.040,47.305,410.439,169.083,40.400,157.580
C04367=1036.047,47.555,410.422,169.085,40.401,157.580
C04368=1036.053,47.804,410.406,169.087,40.401,157.580
C04369=1036.060,48.054,410.388,169.089,40.400,157.580
C04370=1036.065,48.303,410.371,169.091,40.400,157.580
C04371=1036.072,48.552,410.353,169.093,40.400,157.580
C04372=1036.078,48.801,410.337,169.095,40.400,157.580
C04373=1036.084,49.051,410.319,169.097,40.400,157.580
C04374=1036.091,49.300,410.302,169.099,40.399,157.580
C04375=1036.097,49.549,410.286,169.102,40.400,157.581
C04376=1036.103,49.799,410.268,169.104,40.400,157.581
C04377=1036.109,50.048,410.251,169.106,40.399,157.581
C04378=1036.116,50.297,410.234,169.109,40.399,157.581
C04379=1036.122,50.546,410.218,169.111,40.399,157.581
C04380=1036.128,50.796,410.200,169.113,40.399,157.581
C04381=1036.135,51.046,410.182,169.115,40.398,157.581
C04382=1036.141,51.294,410.165,169.117,40.398,157.581
C04383=1036.147,51.545,410.148,169.119,40.398,157.581
C04384=1036.153,51.793,410.131,169.121,40.398,157.581
C04385=1036.160,52.043,410.114,169.123,40.398,157.581
C04386=1036.165,52.292,410.096,169.125,40.398,157.581
C04387=1036.172,52.541,410.079,169.127,40.398,157.581
C04388=1036.179,52.790,410.062,169.129,40.398,157.581
C04389=1036.184,53.040,410.045,169.131,40.397,157.581
C04390=1036.191,53.289,410.028,169.134,40.397,157.582
C04391=1036.197,53.539,410.010,169.136,40.397,157.582
C04392=1036.203,53.788,409.993,169.138,40.397,157.582
C04393=1036.210,54.037,409.975,169.140,40.397,157.582
C04394=1036.217,54.286,409.958,169.142,40.396,157.582
C04395=1036.222,54.536,409.941,169.144,40.397,157.582
C04396=1036.229,54.786,409.924,169.146,40.397,157.582
C04397=1036.235,55.034,409.907,169.148,40.396,157.582
C04398=1036.241,55.284,409.889,169.150,40.396,157.582
C04399=1036.248,55.533,409.872,169.152,40.396,157.582
C04400=1036.254,55.782,409.855,169.154,40.396,157.582
C04401=1036.260,56.032,409.837,169.157,40.395,157.582
C04402=1036.267,56.281,409.820,169.159,40.395,157.582
C04403=1036.273,56.530,409.802,169.161,40.395,157.582
C04404=1036.280,56.780,409.785,169.164,40.395,157.582
C04405=1036.286,57.029,409.768,169.166,40.395,157.582
C04406=1036.293,57.278,409.750,169.168,40.394,157.583
C04407=1036.299,57.528,409.733,169.170,40.394,157.583
C04408=1036.305,57.777,409.716,169.172,40.394,157.583
C04409=1036.312,58.027,409.699,169.174,40.394,157.583
C04410=1036.317,58.276,409.681,169.176,40.394,157.583
C04411=1036.324,58.525,409.664,169.178,40.393,157.583
C04412=1036.330,58.775,409.646,169.181,40.393,157.583
C04413=1036.336,59.023,409.629,169.183,40.393,157.583
C04414=1036.343,59.273,409.612,169.185,40.393,157.583
C04415=1036.349,59.523,409.594,169.187,40.393,157.583
C04416=1036.356,59.771,409.577,169.189,40.393,157.583
C04417=1036.363,60.021,409.559,169.191,40.393,157.583
C04418=1036.370,60.307,409.539,169.193,40.393,157.583
C04419=1036.377,60.593,409.518,169.196,40.392,157.583
C04420=1036.385,60.879,409.498,169.198,40.392,157.583
C04421=1036.392,61.165,409.478,169.201,40.392,157.583
C04422=1036.399,61.415,409.461,169.203,40.392,157.584
C04423=1036.405,61.663,409.444,169.205,40.391,157.584
C04424=1036.411,61.913,409.426,169.207,40.391,157.584
C04425=1036.418,62.163,409.408,169.209,40.391,157.584
C04426=1036.424,62.412,409.391,169.211,40.391,157.584
C04427=1036.430,62.661,409.374,169.213,40.391,157.584
C04428=1036.437,62.911,409.356,169.215,40.390,157.584
C04429=1036.443,63.160,409.338,169.218,40.390,157.584
C04430=1036.450,63.410,409.321,169.220,40.390,157.584
C04431=1036.457,63.658,409.303,169.222,40.390,157.584
C04432=1036.463,63.908,409.285,169.224,40.389,157.584
C04433=1036.469,64.157,409.267,169.226,40.389,157.584
C04434=1036.475,64.406,409.250,169.228,40.389,157.584
C04435=1036.481,64.656,409.232,169.230,40.389,157.584
C04436=1036.488,64.905,409.214,169.232,40.389,157.584
C04437=1036.495,65.154,409.196,169.235,40.389,157.584
C04438=1036.500,65.403,409.179,169.237,40.389,157.585
C04439=1036.506,65.653,409.161,169.239,40.389,157.585
C04440=1036.513,65.902,409.143,169.241,40.388,157.585
C04441=1036.520,66.152,409.125,169.243,40.388,157.585
C04442=1036.525,66.401,409.107,169.245,40.388,157.585
C04443=1036.532,66.650,409.089,169.248,40.388,157.585
C04444=1036.538,66.899,409.071,169.250,40.388,157.585
C04445=1036.544,67.149,409.054,169.252,40.388,157.585
C04446=1036.551,67.398,409.037,169.254,40.388,157.585
C04447=1036.557,67.647,409.018,169.256,40.388,157.585
C04448=1036.563,67.897,409.000,169.258,40.387,157.585
C04449=1036.569,68.146,408.982,169.260,40.387,157.585
C04450=1036.576,68.394,408.964,169.262,40.387,157.585
C04451=1036.582,68.644,408.946,169.264,40.387,157.585
C04452=1036.588,68.894,408.928,169.266,40.387,157.586
C04453=1036.595,69.143,408.910,169.268,40.387,157.586
C04454=1036.601,69.392,408.893,169.270,40.387,157.586
C04455=1036.607,69.641,408.874,169.272,40.387,157.586
C04456=1036.613,69.891,408.856,169.274,40.386,157.586
C04457=1036.620,70.140,408.838,169.276,40.387,157.586
C04458=1036.626,70.390,408.820,169.279,40.387,157.586
C04459=1036.632,70.638,408.803,169.281,40.386,157.586
C04460=1036.639,70.887,408.784,169.284,40.386,157.586
C04461=1036.645,71.137,408.766,169.286,40.386,157.586
C04462=1036.651,71.386,408.747,169.288,40.386,157.586
C04463=1036.657,71.636,408.730,169.290,40.386,157.586
C04464=1036.663,71.884,408.711,169.292,40.386,157.586
C04465=1036.669,72.134,408.693,169.294,40.386,157.586
C04466=1036.676,72.383,408.675,169.296,40.386,157.587
C04467=1036.683,72.633,408.657,169.298,40.386,157.587
C04468=1036.689,72.882,408.639,169.300,40.386,157.587
C04469=1036.695,73.131,408.621,169.302,40.386,157.587
C04470=1036.701,73.380,408.602,169.304,40.385,157.587
C04471=1036.707,73.630,408.585,169.306,40.385,157.587
C04472=1036.713,73.879,408.566,169.308,40.386,157.587
C04473=1036.720,74.129,408.548,169.310,40.385,157.587
C04474=1036.726,74.378,408.529,169.312,40.385,157.587
C04475=1036.732,74.626,408.512,169.314,40.385,157.587
C04476=1036.739,74.876,408.494,169.316,40.385,157.587
C04477=1036.745,75.125,408.475,169.319,40.385,157.587
C04478=1036.751,75.374,408.457,169.321,40.385,157.587
C04479=1036.758,75.624,408.438,169.324,40.385,157.588
C04480=1036.764,75.873,408.421,169.326,40.384,157.588
C04481=1036.770,76.122,408.402,169.328,40.384,157.588
C04482=1036.778,76.408,408.381,169.330,40.384,157.588
C04483=1036.785,76.694,408.360,169.332,40.385,157.588
C04484=1036.792,76.980,408.340,169.335,40.384,157.588
C04485=1036.799,77.266,408.318,169.337,40.384,157.588
C04486=1036.805,77.515,408.299,169.339,40.384,157.588
C04487=1036.812,77.765,408.281,169.341,40.384,157.588
C04488=1036.818,78.014,408.263,169.343,40.384,157.588
C04489=1036.824,78.263,408.244,169.345,40.384,157.588
C04490=1036.830,78.512,408.226,169.347,40.384,157.588
C04491=1036.836,78.762,408.208,169.349,40.384,157.589
C04492=1036.843,79.011,408.189,169.351,40.384,157.589
C04493=1036.849,79.260,408.171,169.353,40.384,157.589
C04494=1036.855,79.500,408.153,169.355,40.383,157.589
C04495=1036.860,79.739,408.135,169.358,40.384,157.589
C04496=1036.867,79.979,408.117,169.360,40.384,157.589
C04497=1036.872,80.218,408.099,169.362,40.384,157.589
C04498=1036.878,80.458,408.081,169.364,40.383,157.589
C04499=1036.885,80.697,408.063,169.366,40.384,157.589
C04500=1036.890,80.936,408.046,169.368,40.384,157.589
C04501=1036.896,81.177,408.028,169.370,40.383,157.589
C04502=1036.903,81.426,408.009,169.372,40.384,157.590
C04503=1036.909,81.675,407.990,169.374,40.384,157.590
C04504=1036.915,81.924,407.971,169.376,40.383,157.590
C04505=1036.921,82.173,407.953,169.378,40.383,157.590
C04506=1036.927,82.423,407.935,169.380,40.384,157.590
C04507=1036.934,82.672,407.916,169.382,40.383,157.590
C04508=1036.940,82.921,407.898,169.384,40.383,157.590
C04509=1036.945,83.170,407.879,169.386,40.383,157.590
C04510=1036.952,83.419,407.860,169.388,40.383,157.590
C04511=1036.958,83.668,407.841,169.390,40.383,157.590
C04512=1036.965,83.917,407.823,169.394,40.383,157.590
C04513=1036.971,84.166,407.804,169.396,40.383,157.590
C04514=1036.977,84.417,407.785,169.398,40.383,157.591
C04515=1036.983,84.666,407.767,169.400,40.383,157.591
C04516=1036.989,84.915,407.748,169.402,40.383,157.591
C04517=1036.996,85.164,407.730,169.404,40.383,157.591
C04518=1037.002,85.413,407.711,169.406,40.383,157.591
C04519=1037.009,85.662,407.692,169.408,40.383,157.591
C04520=1037.014,85.912,407.673,169.410,40.383,157.591
C04521=1037.021,86.161,407.654,169.412,40.382,157.591
C04522=1037.027,86.410,407.636,169.414,40.383,157.591
C04523=1037.034,86.659,407.617,169.416,40.383,157.591
C04524=1037.040,86.908,407.598,169.418,40.382,157.591
C04525=1037.046,87.158,407.579,169.420,40.382,157.591
C04526=1037.052,87.407,407.561,169.422,40.382,157.591
C04527=1037.059,87.656,407.542,169.424,40.382,157.592
C04528=1037.065,87.905,407.523,169.426,40.382,157.592
C04529=1037.072,88.155,407.504,169.429,40.382,157.592
C04530=1037.078,88.404,407.485,169.432,40.382,157.592
C04531=1037.084,88.653,407.466,169.434,40.382,157.592
C04532=1037.091,88.902,407.448,169.436,40.382,157.592
C04533=1037.097,89.152,407.429,169.438,40.382,157.592
C04534=1037.103,89.401,407.410,169.440,40.382,157.592
C04535=1037.109,89.650,407.391,169.442,40.381,157.592
C04536=1037.116,89.899,407.372,169.444,40.382,157.592
C04537=1037.122,90.148,407.354,169.446,40.382,157.592
C04538=1037.128,90.398,407.335,169.448,40.381,157.592
C04539=1037.134,90.646,407.315,169.450,40.382,157.593
C04540=1037.140,90.896,407.296,169.452,40.382,157.593
C04541=1037.146,91.145,407.277,169.454,40.381,157.593
C04542=1037.152,91.394,407.258,169.456,40.382,157.593
C04543=1037.159,91.643,407.239,169.458,40.382,157.593
C04544=1037.165,91.892,407.219,169.460,40.381,157.593
C04545=1037.171,92.141,407.201,169.463,40.382,157.593
C04546=1037.179,92.447,407.177,169.466,40.382,157.593
C04547=1037.186,92.752,407.154,169.468,40.382,157.593
C04548=1037.194,93.058,407.131,169.471,40.382,157.594
C04549=1037.201,93.363,407.107,169.473,40.382,157.594
C04550=1037.207,93.612,407.088,169.475,40.382,157.594
C04551=1037.214,93.861,407.069,169.478,40.382,157.594
C04552=1037.220,94.110,407.049,169.480,40.381,157.594
C04553=1037.226,94.359,407.031,169.482,40.382,157.594
C04554=1037.232,94.609,407.011,169.484,40.382,157.594
C04555=1037.239,94.859,406.992,169.486,40.381,157.594
C04556=1037.245,95.107,406.972,169.488,40.382,157.594
C04557=1037.251,95.356,406.954,169.490,40.382,157.594
C04558=1037.257,95.606,406.934,169.492,40.382,157.594
C04559=1037.264,95.854,406.915,169.495,40.382,157.595
C04560=1037.269,96.104,406.896,169.497,40.382,157.595
C04561=1037.276,96.353,406.877,169.499,40.382,157.595
C04562=1037.282,96.602,406.857,169.501,40.381,157.595
C04563=1037.289,96.852,406.838,169.503,40.382,157.595
C04564=1037.294,97.101,406.819,169.505,40.382,157.595
C04565=1037.301,97.349,406.800,169.507,40.381,157.595
C04566=1037.307,97.599,406.780,169.509,40.382,157.595
C04567=1037.313,97.848,406.762,169.511,40.382,157.595
C04568=1037.320,98.098,406.741,169.514,40.381,157.595
C04569=1037.326,98.347,406.723,169.516,40.382,157.596
C04570=1037.332,98.595,406.703,169.518,40.382,157.596
C04571=1037.339,98.845,406.684,169.520,40.381,157.596
C04572=1037.344,99.094,406.665,169.522,40.381,157.596
C04573=1037.352,99.343,406.645,169.525,40.382,157.596
C04574=1037.357,99.593,406.626,169.527,40.381,157.596
C04575=1037.364,99.841,406.607,169.529,40.381,157.596
C04576=1037.370,100.091,406.587,169.531,40.382,157.596
C04577=1037.375,100.340,406.568,169.533,40.381,157.596
C04578=1037.383,100.589,406.548,169.535,40.381,157.596
C04579=1037.388,100.839,406.529,169.537,40.382,157.596
C04580=1037.394,101.088,406.509,169.539,40.381,157.596
C04581=1037.400,101.336,406.489,169.541,40.382,157.597
C04582=1037.407,101.585,406.470,169.543,40.382,157.597
C04583=1037.413,101.834,406.451,169.546,40.381,157.597
C04584=1037.419,102.084,406.431,169.548,40.382,157.597
C04585=1037.425,102.333,406.411,169.550,40.382,157.597
C04586=1037.431,102.583,406.392,169.553,40.382,157.597
C04587=1037.438,102.831,406.372,169.555,40.382,157.597
C04588=1037.444,103.080,406.352,169.557,40.382,157.597
C04589=1037.450,103.330,406.333,169.559,40.382,157.597
C04590=1037.456,103.579,406.313,169.561,40.382,157.597
C04591=1037.462,103.828,406.294,169.563,40.382,157.598
C04592=1037.468,104.077,406.274,169.565,40.382,157.598
C04593=1037.475,104.326,406.254,169.567,40.382,157.598
C04594=1037.481,104.576,406.235,169.569,40.382,157.598
C04595=1037.487,104.825,406.215,169.571,40.382,157.598
C04596=1037.492,105.074,406.195,169.573,40.383,157.598
C04597=1037.500,105.323,406.176,169.575,40.382,157.598
C04598=1037.506,105.572,406.156,169.578,40.383,157.598
C04599=1037.511,105.821,406.137,169.581,40.382,157.598
C04600=1037.517,106.070,406.117,169.583,40.382,157.599
C04601=1037.524,106.320,406.096,169.585,40.383,157.599
C04602=1037.530,106.569,406.078,169.587,40.382,157.599
C04603=1037.536,106.818,406.058,169.589,40.382,157.599
C04604=1037.542,107.067,406.038,169.591,40.383,157.599
C04605=1037.549,107.316,406.017,169.593,40.383,157.599
C04606=1037.555,107.565,405.998,169.595,40.383,157.599
C04607=1037.561,107.814,405.979,169.597,40.383,157.599
C04608=1037.568,108.064,405.958,169.599,40.383,157.599
C04609=1037.574,108.312,405.938,169.601,40.383,157.600
C04610=1037.581,108.598,405.916,169.604,40.383,157.600
C04611=1037.588,108.884,405.893,169.607,40.383,157.600
C04612=1037.595,109.170,405.870,169.610,40.383,157.600
C04613=1037.602,109.456,405.848,169.612,40.383,157.600
C04614=1037.609,109.705,405.828,169.614,40.383,157.600
C04615=1037.614,109.955,405.808,169.616,40.383,157.600
C04616=1037.620,110.204,405.788,169.618,40.383,157.600
C04617=1037.628,110.453,405.769,169.620,40.383,157.600
C04618=1037.634,110.702,405.749,169.623,40.383,157.600
C04619=1037.640,110.951,405.728,169.625,40.383,157.601
C04620=1037.646,111.200,405.708,169.627,40.383,157.601
C04621=1037.652,111.449,405.689,169.629,40.383,157.601
C04622=1037.659,111.699,405.669,169.631,40.383,157.601
C04623=1037.665,111.948,405.649,169.634,40.383,157.601
C04624=1037.671,112.196,405.629,169.636,40.383,157.601
C04625=1037.677,112.446,405.609,169.638,40.383,157.601
C04626=1037.683,112.695,405.589,169.640,40.384,157.601
C04627=1037.689,112.944,405.569,169.642,40.383,157.601
C04628=1037.696,113.193,405.548,169.644,40.384,157.602
C04629=1037.702,113.442,405.528,169.647,40.384,157.602
C04630=1037.707,113.691,405.508,169.649,40.384,157.602
C04631=1037.714,113.941,405.487,169.651,40.384,157.602
C04632=1037.720,114.189,405.468,169.653,40.384,157.602
C04633=1037.726,114.438,405.448,169.655,40.384,157.602
C04634=1037.731,114.688,405.427,169.658,40.384,157.602
C04635=1037.737,114.937,405.407,169.660,40.385,157.602
C04636=1037.743,115.186,405.387,169.662,40.385,157.603
C04637=1037.750,115.435,405.366,169.664,40.385,157.603
C04638=1037.755,115.684,405.346,169.666,40.385,157.603
C04639=1037.762,115.934,405.326,169.668,40.385,157.603
C04640=1037.768,116.183,405.306,169.670,40.385,157.603
C04641=1037.774,116.431,405.286,169.672,40.386,157.603
C04642=1037.780,116.681,405.265,169.675,40.386,157.603
C04643=1037.786,116.930,405.245,169.677,40.386,157.603
C04644=1037.792,117.178,405.224,169.680,40.386,157.604
C04645=1037.799,117.428,405.204,169.682,40.386,157.604
C04646=1037.804,117.677,405.183,169.684,40.386,157.604
C04647=1037.810,117.926,405.163,169.686,40.386,157.604
C04648=1037.816,118.175,405.143,169.688,40.387,157.604
C04649=1037.822,118.424,405.122,169.690,40.386,157.604
C04650=1037.828,118.674,405.102,169.692,40.387,157.604
C04651=1037.835,118.922,405.081,169.694,40.387,157.604
C04652=1037.841,119.172,405.061,169.697,40.387,157.605
C04653=1037.846,119.421,405.040,169.699,40.388,157.605
C04654=1037.853,119.670,405.020,169.702,40.387,157.605
C04655=1037.859,119.919,405.000,169.704,40.388,157.605
C04656=1037.865,120.167,404.980,169.706,40.387,157.605
C04657=1037.871,120.417,404.959,169.708,40.388,157.605
C04658=1037.877,120.666,404.939,169.710,40.388,157.605
C04659=1037.884,120.915,404.918,169.712,40.388,157.605
C04660=1037.889,121.164,404.898,169.714,40.388,157.605
C04661=1037.896,121.413,404.877,169.716,40.388,157.606
C04662=1037.902,121.662,404.857,169.719,40.388,157.606
C04663=1037.909,121.912,404.836,169.722,40.388,157.606
C04664=1037.914,122.160,404.815,169.724,40.388,157.606
C04665=1037.921,122.410,404.795,169.726,40.389,157.606
C04666=1037.927,122.659,404.775,169.728,40.388,157.606
C04667=1037.933,122.908,404.754,169.730,40.389,157.606
C04668=1037.939,123.157,404.733,169.732,40.389,157.607
C04669=1037.945,123.406,404.713,169.734,40.389,157.607
C04670=1037.951,123.655,404.692,169.736,40.390,157.607
C04671=1037.958,123.904,404.671,169.739,40.389,157.607
C04672=1037.964,124.153,404.651,169.742,40.390,157.607
C04673=1037.970,124.402,404.631,169.744,40.389,157.607
C04674=1037.976,124.688,404.607,169.746,40.390,157.607
C04675=1037.983,124.974,404.583,169.749,40.390,157.607
C04676=1037.991,125.260,404.559,169.751,40.390,157.607
C04677=1037.998,125.546,404.536,169.754,40.390,157.608
C04678=1038.005,125.795,404.515,169.756,40.390,157.608
C04679=1038.011,126.043,404.495,169.758,40.390,157.608
C04680=1038.017,126.293,404.474,169.760,40.390,157.608
C04681=1038.023,126.541,404.454,169.762,40.390,157.608
C04682=1038.029,126.791,404.433,169.765,40.391,157.608
C04683=1038.036,127.040,404.412,169.768,40.390,157.608
C04684=1038.042,127.289,404.392,169.770,40.391,157.608
C04685=1038.048,127.538,404.371,169.772,40.391,157.609
C04686=1038.054,127.787,404.351,169.774,40.391,157.609
C04687=1038.061,128.036,404.329,169.776,40.391,157.609
C04688=1038.067,128.285,404.309,169.778,40.391,157.609
C04689=1038.074,128.533,404.288,169.781,40.391,157.609
C04690=1038.079,128.783,404.267,169.783,40.391,157.609
C04691=1038.085,129.032,404.247,169.785,40.391,157.609
C04692=1038.092,129.281,404.226,169.788,40.392,157.609
C04693=1038.098,129.531,404.205,169.790,40.391,157.609
C04694=1038.104,129.779,404.185,169.793,40.392,157.610
C04695=1038.111,130.029,404.164,169.795,40.391,157.610
C04696=1038.117,130.278,404.143,169.797,40.392,157.610
C04697=1038.124,130.526,404.122,169.799,40.392,157.610
C04698=1038.130,130.775,404.102,169.801,40.392,157.610
C04699=1038.136,131.025,404.080,169.803,40.392,157.610
C04700=1038.142,131.274,404.059,169.806,40.392,157.610
C04701=1038.148,131.523,404.038,169.809,40.393,157.611
C04702=1038.154,131.773,404.017,169.811,40.392,157.611
C04703=1038.160,132.021,403.996,169.813,40.393,157.611
C04704=1038.167,132.270,403.975,169.815,40.393,157.611
C04705=1038.172,132.519,403.955,169.817,40.393,157.611
C04706=1038.179,132.768,403.934,169.820,40.393,157.611
C04707=1038.185,133.017,403.912,169.822,40.394,157.611
C04708=1038.191,133.266,403.891,169.824,40.394,157.611
C04709=1038.197,133.515,403.870,169.826,40.394,157.612
C04710=1038.203,133.764,403.849,169.829,40.395,157.612
C04711=1038.209,134.013,403.827,169.831,40.394,157.612
C04712=1038.216,134.262,403.807,169.834,40.395,157.612
C04713=1038.222,134.512,403.785,169.836,40.395,157.612
C04714=1038.227,134.760,403.764,169.838,40.395,157.612
C04715=1038.234,135.009,403.743,169.840,40.395,157.612
C04716=1038.240,135.259,403.722,169.842,40.396,157.613
C04717=1038.246,135.507,403.701,169.844,40.396,157.613
C04718=1038.252,135.756,403.680,169.848,40.396,157.613
C04719=1038.259,136.005,403.658,169.850,40.396,157.613
C04720=1038.264,136.254,403.637,169.852,40.396,157.613
C04721=1038.271,136.503,403.617,169.854,40.397,157.613
C04722=1038.277,136.753,403.595,169.856,40.396,157.613
C04723=1038.283,137.002,403.573,169.859,40.397,157.614
C04724=1038.289,137.250,403.553,169.861,40.397,157.614
C04725=1038.296,137.499,403.531,169.863,40.397,157.614
C04726=1038.301,137.749,403.510,169.865,40.397,157.614
C04727=1038.307,137.998,403.489,169.868,40.398,157.614
C04728=1038.314,138.246,403.468,169.871,40.397,157.614
C04729=1038.320,138.496,403.446,169.873,40.398,157.614
C04730=1038.326,138.745,403.425,169.875,40.398,157.615
C04731=1038.332,138.993,403.403,169.877,40.399,157.615
C04732=1038.339,139.242,403.382,169.879,40.399,157.615
C04733=1038.345,139.492,403.361,169.882,40.399,157.615
C04734=1038.351,139.741,403.339,169.885,40.399,157.615
C04735=1038.357,139.989,403.318,169.887,40.399,157.615
C04736=1038.363,140.238,403.296,169.889,40.399,157.615
C04737=1038.369,140.488,403.274,169.891,40.400,157.616
C04738=1038.375,140.773,403.250,169.894,40.400,157.616
C04739=1038.383,141.059,403.225,169.896,40.401,157.616
C04740=1038.389,141.345,403.201,169.899,40.401,157.616
C04741=1038.397,141.630,403.176,169.902,40.401,157.616
C04742=1038.403,141.878,403.155,169.905,40.401,157.616
C04743=1038.409,142.128,403.134,169.907,40.402,157.617
C04744=1038.415,142.377,403.112,169.909,40.402,157.617
C04745=1038.421,142.626,403.090,169.911,40.402,157.617
C04746=1038.427,142.875,403.069,169.913,40.402,157.617
C04747=1038.433,143.124,403.047,169.916,40.403,157.617
C04748=1038.439,143.373,403.026,169.919,40.403,157.617
C04749=1038.446,143.622,403.003,169.921,40.403,157.617
C04750=1038.452,143.871,402.982,169.923,40.403,157.618
C04751=1038.457,144.119,402.961,169.926,40.403,157.618
C04752=1038.464,144.369,402.939,169.928,40.404,157.618
C04753=1038.470,144.618,402.917,169.930,40.404,157.618
C04754=1038.476,144.867,402.896,169.932,40.404,157.618
C04755=1038.483,145.116,402.875,169.935,40.404,157.618
C04756=1038.489,145.365,402.853,169.938,40.405,157.619
C04757=1038.495,145.613,402.831,169.940,40.405,157.619
C04758=1038.501,145.862,402.809,169.942,40.405,157.619
C04759=1038.507,146.111,402.788,169.944,40.406,157.619
C04760=1038.513,146.361,402.766,169.947,40.406,157.619
C04761=1038.519,146.610,402.744,169.949,40.406,157.619
C04762=1038.526,146.859,402.723,169.951,40.406,157.620
C04763=1038.532,147.108,402.700,169.954,40.407,157.620
C04764=1038.538,147.357,402.679,169.957,40.407,157.620
C04765=1038.544,147.605,402.658,169.959,40.407,157.620
C04766=1038.550,147.854,402.636,169.961,40.408,157.620
C04767=1038.556,148.103,402.613,169.963,40.407,157.620
C04768=1038.562,148.353,402.591,169.966,40.408,157.621
C04769=1038.568,148.602,402.570,169.968,40.408,157.621
C04770=1038.575,148.850,402.547,169.971,40.409,157.621
C04771=1038.581,149.100,402.526,169.973,40.409,157.621
C04772=1038.587,149.349,402.504,169.976,40.409,157.621
C04773=1038.593,149.597,402.482,169.978,40.409,157.621
C04774=1038.599,149.846,402.460,169.980,40.410,157.621
C04775=1038.604,150.095,402.438,169.982,40.410,157.622
C04776=1038.611,150.344,402.416,169.986,40.410,157.622
C04777=1038.617,150.593,402.394,169.988,40.411,157.622
C04778=1038.623,150.842,402.372,169.990,40.411,157.622
C04779=1038.630,151.091,402.350,169.993,40.412,157.622
C04780=1038.635,151.340,402.328,169.995,40.412,157.623
C04781=1038.641,151.589,402.306,169.997,40.412,157.623
C04782=1038.648,151.838,402.284,169.999,40.412,157.623
C04783=1038.654,152.087,402.262,170.003,40.413,157.623
C04784=1038.660,152.335,402.240,170.005,40.413,157.623
C04785=1038.665,152.584,402.217,170.007,40.413,157.623
C04786=1038.672,152.833,402.196,170.009,40.414,157.624
C04787=1038.678,153.083,402.174,170.012,40.414,157.624
C04788=1038.684,153.331,402.152,170.014,40.415,157.624
C04789=1038.690,153.580,402.130,170.016,40.414,157.624
C04790=1038.696,153.829,402.107,170.020,40.415,157.624
C04791=1038.702,154.079,402.086,170.022,40.415,157.624
C04792=1038.709,154.327,402.063,170.024,40.416,157.625
C04793=1038.715,154.576,402.042,170.026,40.416,157.625
C04794=1038.721,154.825,402.019,170.029,40.416,157.625
C04795=1038.727,155.074,401.996,170.032,40.417,157.625
C04796=1038.733,155.323,401.974,170.034,40.417,157.625
C04797=1038.739,155.572,401.952,170.037,40.417,157.626
C04798=1038.745,155.821,401.930,170.039,40.418,157.626
C04799=1038.751,156.070,401.907,170.041,40.418,157.626
C04800=1038.757,156.319,401.885,170.043,40.419,157.626
C04801=1038.764,156.568,401.863,170.047,40.419,157.626
C04802=1038.771,156.853,401.837,170.049,40.419,157.626
C04803=1038.778,157.138,401.812,170.052,40.420,157.627
C04804=1038.784,157.424,401.786,170.055,40.420,157.627
C04805=1038.791,157.709,401.761,170.057,40.421,157.627
C04806=1038.797,157.957,401.738,170.060,40.421,157.627
C04807=1038.804,158.206,401.716,170.063,40.421,157.627
C04808=1038.809,158.455,401.694,170.065,40.422,157.628
C04809=1038.816,158.704,401.671,170.068,40.422,157.628
C04810=1038.822,158.952,401.649,170.070,40.422,157.628
C04811=1038.828,159.203,401.626,170.072,40.423,157.628
C04812=1038.835,159.451,401.604,170.076,40.423,157.628
C04813=1038.840,159.700,401.581,170.078,40.424,157.629
C04814=1038.847,159.949,401.559,170.080,40.424,157.629
C04815=1038.853,160.198,401.537,170.083,40.424,157.629
C04816=1038.859,160.447,401.514,170.085,40.425,157.629
C04817=1038.865,160.696,401.491,170.087,40.425,157.629
C04818=1038.870,160.945,401.468,170.090,40.426,157.630
C04819=1038.876,161.194,401.445,170.093,40.426,157.630
C04820=1038.882,161.442,401.423,170.095,40.427,157.630
C04821=1038.888,161.691,401.400,170.097,40.427,157.630
C04822=1038.894,161.940,401.377,170.100,40.428,157.630
C04823=1038.899,162.189,401.355,170.103,40.428,157.631
C04824=1038.906,162.438,401.332,170.105,40.429,157.631
C04825=1038.912,162.687,401.309,170.108,40.429,157.631
C04826=1038.917,162.936,401.287,170.110,40.430,157.631
C04827=1038.923,163.185,401.264,170.112,40.430,157.632
C04828=1038.929,163.434,401.241,170.115,40.431,157.632
C04829=1038.935,163.682,401.218,170.118,40.431,157.632
C04830=1038.941,163.931,401.195,170.120,40.432,157.632
C04831=1038.947,164.180,401.172,170.122,40.433,157.632
C04832=1038.952,164.429,401.149,170.125,40.433,157.633
C04833=1038.959,164.679,401.126,170.128,40.433,157.633
C04834=1038.965,164.927,401.104,170.130,40.434,157.633
C04835=1038.971,165.176,401.081,170.133,40.434,157.633
C04836=1038.977,165.425,401.058,170.135,40.435,157.633
C04837=1038.982,165.674,401.035,170.137,40.436,157.634
C04838=1038.988,165.922,401.011,170.141,40.436,157.634
C04839=1038.995,166.171,400.989,170.143,40.436,157.634
C04840=1039.001,166.420,400.966,170.145,40.437,157.634
C04841=1039.006,166.668,400.943,170.148,40.437,157.634
C04842=1039.013,166.918,400.920,170.151,40.438,157.635
C04843=1039.018,167.167,400.897,170.154,40.438,157.635
C04844=1039.025,167.416,400.874,170.156,40.439,157.635
C04845=1039.031,167.664,400.851,170.158,40.439,157.635
C04846=1039.036,167.913,400.829,170.161,40.440,157.636
C04847=1039.042,168.162,400.805,170.164,40.441,157.636
C04848=1039.049,168.411,400.782,170.166,40.441,157.636
C04849=1039.055,168.660,400.759,170.169,40.441,157.636
C04850=1039.061,168.909,400.736,170.171,40.442,157.636
C04851=1039.067,169.158,400.713,170.173,40.442,157.637
C04852=1039.072,169.406,400.690,170.177,40.443,157.637
C04853=1039.079,169.655,400.666,170.179,40.444,157.637
C04854=1039.085,169.904,400.643,170.182,40.444,157.637
C04855=1039.091,170.153,400.621,170.184,40.444,157.638
C04856=1039.097,170.402,400.598,170.186,40.445,157.638
C04857=1039.103,170.650,400.574,170.190,40.446,157.638
C04858=1039.109,170.900,400.551,170.192,40.446,157.638
C04859=1039.115,171.149,400.528,170.195,40.446,157.638
C04860=1039.121,171.397,400.505,170.197,40.447,157.639
C04861=1039.128,171.645,400.482,170.199,40.448,157.639
C04862=1039.134,171.895,400.459,170.203,40.448,157.639
C04863=1039.140,172.144,400.436,170.205,40.449,157.639
C04864=1039.145,172.393,400.413,170.208,40.449,157.640
C04865=1039.151,172.641,400.389,170.210,40.450,157.640
C04866=1039.159,172.926,400.363,170.214,40.450,157.640
C04867=1039.166,173.211,400.336,170.217,40.451,157.640
C04868=1039.173,173.496,400.310,170.220,40.452,157.641
C04869=1039.180,173.780,400.283,170.222,40.452,157.641
C04870=1039.186,174.029,400.260,170.225,40.452,157.641
C04871=1039.191,174.278,400.237,170.228,40.453,157.641
C04872=1039.199,174.527,400.214,170.231,40.454,157.641
C04873=1039.204,174.776,400.191,170.233,40.454,157.642
C04874=1039.210,175.024,400.167,170.236,40.454,157.642
C04875=1039.217,175.274,400.144,170.239,40.456,157.642
C04876=1039.223,175.523,400.121,170.241,40.456,157.642
C04877=1039.229,175.771,400.097,170.244,40.456,157.643
C04878=1039.235,176.020,400.074,170.246,40.457,157.643
C04879=1039.241,176.269,400.050,170.249,40.458,157.643
C04880=1039.248,176.518,400.027,170.252,40.458,157.643
C04881=1039.254,176.766,400.004,170.255,40.458,157.643
C04882=1039.260,177.015,399.981,170.257,40.459,157.644
C04883=1039.266,177.264,399.957,170.260,40.460,157.644
C04884=1039.272,177.513,399.934,170.262,40.460,157.644
C04885=1039.279,177.762,399.910,170.266,40.460,157.644
C04886=1039.284,178.011,399.887,170.268,40.461,157.645
C04887=1039.291,178.259,399.863,170.271,40.462,157.645
C04888=1039.298,178.508,399.840,170.273,40.462,157.645
C04889=1039.304,178.757,399.817,170.277,40.463,157.645
C04890=1039.310,179.006,399.793,170.279,40.463,157.645
C04891=1039.316,179.255,399.770,170.282,40.464,157.646
C04892=1039.323,179.504,399.746,170.284,40.464,157.646
C04893=1039.328,179.753,399.723,170.287,40.465,157.646
C04894=1039.334,180.001,399.699,170.290,40.466,157.647
C04895=1039.341,180.250,399.676,170.293,40.466,157.647
C04896=1039.347,180.499,399.652,170.295,40.466,157.647
C04897=1039.353,180.748,399.628,170.298,40.467,157.647
C04898=1039.360,180.996,399.606,170.301,40.468,157.647
C04899=1039.367,181.245,399.582,170.304,40.468,157.648
C04900=1039.373,181.493,399.558,170.306,40.468,157.648
C04901=1039.379,181.743,399.535,170.309,40.469,157.648
C04902=1039.385,181.991,399.511,170.312,40.470,157.648
C04903=1039.392,182.240,399.487,170.315,40.470,157.649
C04904=1039.397,182.489,399.464,170.318,40.470,157.649
C04905=1039.404,182.738,399.440,170.320,40.472,157.649
C04906=1039.410,182.986,399.416,170.323,40.472,157.649
C04907=1039.416,183.236,399.393,170.325,40.472,157.649
C04908=1039.422,183.484,399.369,170.329,40.473,157.650
C04909=1039.429,183.733,399.345,170.331,40.474,157.650
C04910=1039.435,183.982,399.322,170.334,40.475,157.650
C04911=1039.441,184.231,399.297,170.336,40.475,157.651
C04912=1039.447,184.479,399.274,170.340,40.476,157.651
C04913=1039.453,184.728,399.249,170.342,40.477,157.651
C04914=1039.459,184.977,399.225,170.345,40.477,157.651
C04915=1039.465,185.226,399.201,170.348,40.478,157.652
C04916=1039.471,185.474,399.177,170.351,40.479,157.652
C04917=1039.476,185.723,399.153,170.353,40.480,157.652
C04918=1039.483,185.972,399.129,170.356,40.481,157.653
C04919=1039.488,186.220,399.104,170.359,40.481,157.653
C04920=1039.495,186.469,399.080,170.362,40.482,157.653
C04921=1039.500,186.718,399.056,170.364,40.483,157.653
C04922=1039.507,186.967,399.032,170.368,40.483,157.654
C04923=1039.512,187.216,399.008,170.370,40.484,157.654
C04924=1039.519,187.465,398.984,170.373,40.485,157.654
C04925=1039.524,187.713,398.960,170.375,40.486,157.654
C04926=1039.531,187.962,398.936,170.379,40.487,157.655
C04927=1039.536,188.211,398.911,170.382,40.488,157.655
C04928=1039.542,188.460,398.887,170.384,40.488,157.655
C04929=1039.548,188.709,398.863,170.388,40.489,157.656
C04930=1039.555,188.993,398.835,170.391,40.490,157.656
C04931=1039.562,189.277,398.808,170.393,40.491,157.656
C04932=1039.570,189.562,398.779,170.397,40.492,157.657
C04933=1039.576,189.846,398.752,170.400,40.492,157.657
C04934=1039.582,190.095,398.728,170.403,40.493,157.657
C04935=1039.588,190.343,398.703,170.405,40.494,157.658
C04936=1039.594,190.592,398.679,170.409,40.494,157.658
C04937=1039.601,190.841,398.655,170.412,40.495,157.658
C04938=1039.606,191.090,398.631,170.414,40.496,157.658
C04939=1039.613,191.339,398.607,170.417,40.497,157.659
C04940=1039.618,191.586,398.582,170.420,40.498,157.659
C04941=1039.625,191.835,398.558,170.423,40.499,157.659
C04942=1039.631,192.085,398.533,170.426,40.500,157.660
C04943=1039.637,192.333,398.509,170.429,40.500,157.660
C04944=1039.643,192.582,398.485,170.432,40.501,157.660
C04945=1039.650,192.831,398.460,170.434,40.502,157.660
C04946=1039.655,193.079,398.436,170.437,40.502,157.661
C04947=1039.662,193.328,398.412,170.441,40.503,157.661
C04948=1039.668,193.577,398.386,170.443,40.504,157.661
C04949=1039.673,193.825,398.362,170.446,40.505,157.662
C04950=1039.680,194.074,398.338,170.449,40.506,157.662
C04951=1039.686,194.323,398.313,170.452,40.507,157.662
C04952=1039.692,194.571,398.289,170.455,40.507,157.663
C04953=1039.698,194.821,398.264,170.457,40.508,157.663
C04954=1039.705,195.069,398.240,170.461,40.509,157.663
C04955=1039.711,195.318,398.215,170.464,40.510,157.663
C04956=1039.717,195.567,398.191,170.466,40.511,157.664
C04957=1039.723,195.815,398.166,170.470,40.511,157.664
C04958=1039.730,196.064,398.142,170.473,40.512,157.664
C04959=1039.735,196.312,398.117,170.475,40.513,157.665
C04960=1039.742,196.561,398.093,170.479,40.514,157.665
C04961=1039.748,196.811,398.068,170.481,40.514,157.665
C04962=1039.754,197.059,398.043,170.484,40.515,157.665
C04963=1039.760,197.307,398.019,170.488,40.516,157.666
C04964=1039.766,197.556,397.994,170.490,40.517,157.666
C04965=1039.773,197.805,397.970,170.493,40.518,157.666
C04966=1039.779,198.054,397.945,170.496,40.519,157.667
C04967=1039.786,198.303,397.921,170.500,40.519,157.667
C04968=1039.791,198.551,397.896,170.502,40.521,157.667
C04969=1039.797,198.800,397.871,170.505,40.521,157.668
C04970=1039.804,199.048,397.846,170.509,40.522,157.668
C04971=1039.810,199.298,397.822,170.511,40.523,157.668
C04972=1039.817,199.546,397.797,170.514,40.524,157.669
C04973=1039.823,199.795,397.772,170.518,40.525,157.669
C04974=1039.829,200.043,397.748,170.520,40.526,157.669
C04975=1039.835,200.292,397.723,170.523,40.526,157.669
C04976=1039.841,200.541,397.698,170.526,40.527,157.670
C04977=1039.848,200.789,397.673,170.530,40.528,157.670
C04978=1039.855,201.038,397.648,170.532,40.529,157.670
C04979=1039.860,201.287,397.623,170.535,40.530,157.671
C04980=1039.867,201.536,397.598,170.539,40.531,157.671
C04981=1039.872,201.784,397.573,170.541,40.532,157.671
C04982=1039.879,202.033,397.549,170.544,40.533,157.672
C04983=1039.885,202.282,397.524,170.548,40.534,157.672
C04984=1039.891,202.530,397.498,170.550,40.535,157.672
C04985=1039.897,202.779,397.473,170.553,40.536,157.673
C04986=1039.904,203.028,397.448,170.557,40.537,157.673
C04987=1039.909,203.276,397.423,170.559,40.538,157.673
C04988=1039.915,203.525,397.398,170.562,40.538,157.674
C04989=1039.921,203.773,397.373,170.566,40.539,157.674
C04990=1039.928,204.022,397.347,170.569,40.540,157.674
C04991=1039.934,204.271,397.322,170.571,40.541,157.675
C04992=1039.940,204.519,397.297,170.575,40.542,157.675
C04993=1039.946,204.769,397.272,170.578,40.543,157.675
C04994=1039.972,205.819,397.166,170.868,40.647,157.710
C04995=1039.981,206.126,397.134,170.870,40.649,157.711
C04996=1039.989,206.433,397.100,170.873,40.651,157.712
C04997=1039.997,206.740,397.068,170.876,40.653,157.712
C04998=1040.006,207.047,397.035,170.878,40.655,157.713
C04999=1040.013,207.296,397.009,170.881,40.657,157.713
C05000=1040.019,207.544,396.983,170.883,40.659,157.714
C05001=1040.026,207.793,396.956,170.885,40.661,157.714
C05002=1040.032,208.041,396.930,170.887,40.662,157.715
C05003=1040.039,208.290,396.903,170.890,40.664,157.715
C05004=1040.045,208.537,396.876,170.892,40.666,157.715
C05005=1040.052,208.786,396.850,170.894,40.667,157.716
C05006=1040.059,209.035,396.823,170.896,40.669,157.716
C05007=1040.065,209.283,396.797,170.899,40.671,157.717
C05008=1040.072,209.532,396.770,170.901,40.672,157.717
C05009=1040.079,209.781,396.744,170.903,40.675,157.718
C05010=1040.085,210.029,396.717,170.905,40.676,157.718
C05011=1040.092,210.278,396.691,170.908,40.678,157.719
C05012=1040.099,210.525,396.664,170.910,40.680,157.719
C05013=1040.106,210.774,396.637,170.912,40.681,157.720
C05014=1040.113,211.023,396.611,170.914,40.683,157.720
C05015=1040.119,211.271,396.584,170.917,40.685,157.721
C05016=1040.126,211.520,396.557,170.919,40.686,157.721
C05017=1040.133,211.768,396.530,170.921,40.688,157.721
C05018=1040.139,212.017,396.504,170.923,40.690,157.722
C05019=1040.146,212.265,396.477,170.926,40.692,157.723
C05020=1040.152,212.514,396.451,170.928,40.694,157.723
C05021=1040.158,212.762,396.423,170.930,40.695,157.723
C05022=1040.165,213.011,396.396,170.932,40.697,157.724
C05023=1040.171,213.259,396.370,170.935,40.699,157.724
C05024=1040.179,213.508,396.343,170.938,40.701,157.725
C05025=1040.185,213.757,396.316,170.940,40.702,157.725
C05026=1040.191,214.005,396.290,170.942,40.704,157.726
C05027=1040.198,214.253,396.262,170.944,40.706,157.726
C05028=1040.205,214.502,396.235,170.947,40.707,157.727
C05029=1040.211,214.750,396.209,170.949,40.709,157.727
C05030=1040.218,214.998,396.182,170.952,40.711,157.728
C05031=1040.225,215.247,396.155,170.953,40.712,157.728
C05032=1040.231,215.495,396.127,170.956,40.715,157.729
C05033=1040.238,215.744,396.101,170.958,40.716,157.729
C05034=1040.244,215.993,396.074,170.961,40.718,157.730
C05035=1040.252,216.241,396.047,170.963,40.720,157.730
C05036=1040.258,216.489,396.020,170.965,40.721,157.731
C05037=1040.265,216.738,395.993,170.967,40.723,157.731
C05038=1040.271,216.987,395.966,170.970,40.725,157.732
C05039=1040.278,217.235,395.938,170.972,40.726,157.732
C05040=1040.285,217.483,395.912,170.975,40.729,157.733
C05041=1040.291,217.732,395.884,170.977,40.730,157.733
C05042=1040.298,217.980,395.858,170.979,40.732,157.733
C05043=1040.305,218.229,395.830,170.981,40.734,157.734
C05044=1040.312,218.477,395.804,170.984,40.735,157.734
C05045=1040.318,218.725,395.776,170.986,40.737,157.735
C05046=1040.325,218.974,395.749,170.989,40.738,157.735
C05047=1040.332,219.222,395.722,170.991,40.740,157.736
C05048=1040.338,219.471,395.695,170.994,40.742,157.736
C05049=1040.345,219.719,395.669,170.996,40.743,157.737
C05050=1040.352,219.968,395.642,170.998,40.745,157.737
C05051=1040.360,220.280,395.607,171.002,40.747,157.738
C05052=1040.368,220.593,395.573,171.004,40.749,157.738
C05053=1040.376,220.906,395.539,171.007,40.752,157.739
C05054=1040.385,221.218,395.504,171.011,40.754,157.740
C05055=1040.391,221.467,395.476,171.013,40.756,157.740
C05056=1040.397,221.714,395.449,171.015,40.758,157.741
C05057=1040.405,221.963,395.423,171.017,40.759,157.741
C05058=1040.411,222.211,395.395,171.020,40.761,157.742
C05059=1040.418,222.460,395.367,171.022,40.763,157.742
C05060=1040.425,222.708,395.339,171.025,40.765,157.743
C05061=1040.430,222.957,395.313,171.027,40.767,157.743
C05062=1040.437,223.205,395.285,171.030,40.768,157.744
C05063=1040.445,223.453,395.258,171.032,40.770,157.744
C05064=1040.451,223.702,395.230,171.035,40.771,157.745
C05065=1040.458,223.951,395.203,171.036,40.773,157.745
C05066=1040.464,224.199,395.175,171.039,40.775,157.746
C05067=1040.471,224.448,395.148,171.042,40.777,157.746
C05068=1040.477,224.695,395.120,171.044,40.779,157.747
C05069=1040.484,224.944,395.093,171.047,40.780,157.747
C05070=1040.491,225.192,395.066,171.049,40.782,157.747
C05071=1040.497,225.441,395.038,171.052,40.784,157.748
C05072=1040.504,225.689,395.011,171.054,40.785,157.748
C05073=1040.511,225.938,394.983,171.057,40.787,157.749
C05074=1040.518,226.186,394.955,171.059,40.789,157.749
C05075=1040.524,226.435,394.928,171.062,40.791,157.750
C05076=1040.530,226.683,394.900,171.064,40.792,157.750
C05077=1040.537,226.931,394.872,171.067,40.794,157.751
C05078=1040.544,227.179,394.845,171.069,40.795,157.751
C05079=1040.551,227.428,394.818,171.072,40.797,157.752
C05080=1040.557,227.677,394.791,171.074,40.799,157.752
C05081=1040.564,227.925,394.763,171.076,40.801,157.753
C05082=1040.571,228.174,394.735,171.078,40.803,157.753
C05083=1040.577,228.422,394.707,171.081,40.804,157.754
C05084=1040.584,228.670,394.680,171.083,40.806,157.754
C05085=1040.591,228.919,394.652,171.086,40.808,157.755
C05086=1040.598,229.167,394.624,171.089,40.810,157.755
C05087=1040.604,229.416,394.596,171.091,40.811,157.756
C05088=1040.611,229.664,394.569,171.094,40.813,157.756
C05089=1040.618,229.912,394.540,171.096,40.815,157.757
C05090=1040.624,230.160,394.513,171.099,40.816,157.757
C05091=1040.630,230.408,394.485,171.101,40.819,157.758
C05092=1040.637,230.657,394.457,171.104,40.820,157.758
C05093=1040.643,230.905,394.429,171.106,40.822,157.759
C05094=1040.650,231.154,394.401,171.109,40.823,157.759
C05095=1040.657,231.402,394.374,171.112,40.826,157.760
C05096=1040.663,231.651,394.346,171.114,40.827,157.760
C05097=1040.670,231.899,394.318,171.117,40.829,157.761
C05098=1040.677,232.147,394.290,171.119,40.830,157.761
C05099=1040.683,232.396,394.261,171.122,40.832,157.762
C05100=1040.690,232.644,394.234,171.124,40.834,157.762
C05101=1040.696,232.893,394.206,171.127,40.836,157.763
C05102=1040.703,233.140,394.178,171.129,40.838,157.763
C05103=1040.709,233.389,394.149,171.132,40.840,157.764
C05104=1040.716,233.638,394.122,171.134,40.841,157.764
C05105=1040.723,233.886,394.094,171.137,40.843,157.765
C05106=1040.730,234.134,394.065,171.139,40.845,157.765
C05107=1040.738,234.440,394.031,171.143,40.847,157.766
C05108=1040.745,234.744,393.997,171.146,40.849,157.766
C05109=1040.754,235.049,393.962,171.149,40.851,157.767
C05110=1040.762,235.355,393.927,171.152,40.853,157.768
C05111=1040.769,235.603,393.899,171.155,40.855,157.768
C05112=1040.776,235.851,393.871,171.157,40.857,157.769
C05113=1040.781,236.100,393.842,171.160,40.859,157.769
C05114=1040.788,236.348,393.815,171.162,40.860,157.770
C05115=1040.795,236.596,393.786,171.165,40.862,157.770
C05116=1040.802,236.844,393.758,171.168,40.864,157.771
C05117=1040.808,237.093,393.730,171.170,40.866,157.771
C05118=1040.815,237.341,393.702,171.173,40.867,157.772
C05119=1040.821,237.589,393.674,171.176,40.869,157.772
C05120=1040.828,237.837,393.645,171.179,40.871,157.773
C05121=1040.834,238.086,393.617,171.181,40.873,157.773
C05122=1040.841,238.334,393.589,171.184,40.874,157.774
C05123=1040.849,238.583,393.561,171.186,40.876,157.774
C05124=1040.855,238.831,393.532,171.189,40.878,157.775
C05125=1040.862,239.079,393.504,171.192,40.880,157.775
C05126=1040.868,239.328,393.475,171.194,40.881,157.776
C05127=1040.874,239.576,393.447,171.197,40.883,157.776
C05128=1040.881,239.824,393.419,171.199,40.885,157.777
C05129=1040.887,240.073,393.390,171.202,40.887,157.777
C05130=1040.894,240.320,393.362,171.205,40.888,157.778
C05131=1040.902,240.570,393.334,171.208,40.890,157.778
C05132=1040.908,240.818,393.305,171.210,40.892,157.779
C05133=1040.915,241.066,393.277,171.213,40.894,157.779
C05134=1040.921,241.314,393.248,171.215,40.895,157.780
C05135=1040.928,241.562,393.219,171.218,40.898,157.780
C05136=1040.934,241.810,393.190,171.221,40.899,157.781
C05137=1040.941,242.059,393.163,171.223,40.901,157.781
C05138=1040.948,242.308,393.133,171.226,40.903,157.782
C05139=1040.955,242.555,393.105,171.228,40.905,157.782
C05140=1040.961,242.804,393.077,171.232,40.906,157.783
C05141=1040.967,243.052,393.048,171.235,40.908,157.784
C05142=1040.974,243.300,393.019,171.237,40.910,157.784
C05143=1040.980,243.548,392.990,171.240,40.912,157.784
C05144=1040.987,243.797,392.962,171.242,40.914,157.785
C05145=1040.994,244.045,392.933,171.245,40.916,157.786
C05146=1041.000,244.294,392.904,171.247,40.917,157.786
C05147=1041.007,244.541,392.875,171.251,40.919,157.787
C05148=1041.013,244.790,392.847,171.253,40.921,157.787
C05149=1041.020,245.039,392.818,171.256,40.922,157.788
C05150=1041.027,245.287,392.789,171.259,40.925,157.788
C05151=1041.033,245.535,392.760,171.261,40.926,157.789
C05152=1041.039,245.783,392.731,171.264,40.928,157.789
C05153=1041.045,246.031,392.702,171.266,40.930,157.790
C05154=1041.052,246.279,392.674,171.269,40.932,157.790
C05155=1041.059,246.528,392.644,171.273,40.934,157.791
C05156=1041.065,246.776,392.615,171.275,40.936,157.791
C05157=1041.072,247.024,392.586,171.278,40.938,157.792
C05158=1041.078,247.272,392.557,171.280,40.939,157.792
C05159=1041.084,247.520,392.528,171.283,40.941,157.793
C05160=1041.091,247.769,392.499,171.286,40.943,157.793
C05161=1041.098,248.017,392.470,171.289,40.945,157.794
C05162=1041.104,248.265,392.441,171.292,40.947,157.795
C05163=1041.112,248.565,392.405,171.294,40.949,157.795
C05164=1041.120,248.864,392.371,171.298,40.952,157.796
C05165=1041.128,249.163,392.336,171.302,40.954,157.797
C05166=1041.136,249.462,392.301,171.305,40.956,157.797
C05167=1041.143,249.711,392.272,171.307,40.958,157.798
C05168=1041.149,249.959,392.243,171.311,40.960,157.798
C05169=1041.155,250.207,392.214,171.313,40.961,157.799
C05170=1041.161,250.455,392.185,171.316,40.963,157.799
C05171=1041.168,250.704,392.155,171.319,40.965,157.800
C05172=1041.175,250.951,392.125,171.321,40.967,157.801
C05173=1041.182,251.199,392.097,171.325,40.969,157.801
C05174=1041.189,251.448,392.067,171.327,40.970,157.801
C05175=1041.195,251.696,392.038,171.330,40.973,157.802
C05176=1041.201,251.944,392.009,171.333,40.974,157.803
C05177=1041.208,252.193,391.980,171.336,40.976,157.803
C05178=1041.214,252.441,391.950,171.339,40.978,157.804
C05179=1041.221,252.689,391.921,171.341,40.980,157.804
C05180=1041.228,252.938,391.892,171.344,40.982,157.805
C05181=1041.234,253.186,391.863,171.348,40.984,157.805
C05182=1041.241,253.433,391.834,171.350,40.985,157.806
C05183=1041.248,253.682,391.804,171.353,40.987,157.806
C05184=1041.254,253.930,391.775,171.355,40.989,157.807
C05185=1041.261,254.179,391.746,171.359,40.991,157.807
C05186=1041.268,254.426,391.716,171.362,40.993,157.808
C05187=1041.274,254.674,391.687,171.364,40.994,157.809
C05188=1041.281,254.923,391.658,171.367,40.997,157.809
C05189=1041.287,255.171,391.628,171.370,40.998,157.810
C05190=1041.294,255.420,391.598,171.373,41.000,157.810
C05191=1041.300,255.668,391.569,171.376,41.002,157.811
C05192=1041.307,255.916,391.539,171.379,41.003,157.811
C05193=1041.314,256.164,391.511,171.382,41.006,157.812
C05194=1041.321,256.411,391.481,171.384,41.007,157.812
C05195=1041.328,256.660,391.452,171.388,41.009,157.813
C05196=1041.334,256.908,391.423,171.390,41.011,157.813
C05197=1041.341,257.156,391.392,171.393,41.013,157.814
C05198=1041.348,257.405,391.363,171.397,41.015,157.815
C05199=1041.355,257.653,391.333,171.399,41.017,157.815
C05200=1041.361,257.901,391.304,171.402,41.018,157.816
C05201=1041.368,258.149,391.274,171.404,41.020,157.816
C05202=1041.374,258.397,391.245,171.408,41.022,157.817
C05203=1041.382,258.646,391.215,171.411,41.024,157.817
C05204=1041.388,258.894,391.186,171.414,41.026,157.818
C05205=1041.395,259.142,391.156,171.417,41.027,157.818
C05206=1041.402,259.390,391.127,171.420,41.029,157.819
C05207=1041.409,259.638,391.097,171.423,41.031,157.819
C05208=1041.416,259.887,391.068,171.426,41.033,157.820
C05209=1041.422,260.134,391.038,171.428,41.035,157.821
C05210=1041.429,260.383,391.009,171.432,41.037,157.821
C05211=1041.436,260.631,390.979,171.435,41.038,157.822
C05212=1041.443,260.879,390.949,171.437,41.040,157.822
C05213=1041.449,261.127,390.920,171.441,41.042,157.823
C05214=1041.456,261.375,390.890,171.443,41.044,157.823
C05215=1041.463,261.624,390.860,171.447,41.046,157.824
C05216=1041.470,261.871,390.830,171.450,41.047,157.824
C05217=1041.477,262.120,390.800,171.452,41.050,157.825
C05218=1041.484,262.367,390.771,171.456,41.051,157.826
C05219=1041.491,262.665,390.735,171.460,41.054,157.826
C05220=1041.499,262.963,390.699,171.462,41.056,157.827
C05221=1041.507,263.261,390.662,171.466,41.058,157.828
C05222=1041.515,263.559,390.626,171.470,41.061,157.828
C05223=1041.521,263.807,390.597,171.473,41.062,157.829
C05224=1041.529,264.055,390.566,171.476,41.064,157.829
C05225=1041.535,264.303,390.536,171.479,41.066,157.830
C05226=1041.541,264.551,390.507,171.482,41.068,157.831
C05227=1041.548,264.800,390.477,171.485,41.070,157.831
C05228=1041.554,265.047,390.446,171.488,41.072,157.832
C05229=1041.561,265.296,390.416,171.491,41.074,157.832
C05230=1041.569,265.544,390.386,171.494,41.076,157.833
C05231=1041.574,265.792,390.356,171.498,41.078,157.834
C05232=1041.582,266.040,390.325,171.500,41.080,157.834
C05233=1041.588,266.287,390.296,171.504,41.082,157.835
C05234=1041.595,266.536,390.265,171.506,41.083,157.835
C05235=1041.602,266.784,390.235,171.509,41.085,157.836
C05236=1041.608,267.032,390.205,171.513,41.088,157.836
C05237=1041.615,267.280,390.174,171.515,41.089,157.837
C05238=1041.622,267.528,390.144,171.519,41.091,157.838
C05239=1041.628,267.776,390.114,171.522,41.093,157.838
C05240=1041.635,268.024,390.084,171.525,41.095,157.839
C05241=1041.642,268.273,390.054,171.528,41.097,157.839
C05242=1041.648,268.521,390.023,171.531,41.099,157.840
C05243=1041.655,268.769,389.993,171.534,41.101,157.841
C05244=1041.662,269.017,389.962,171.537,41.103,157.841
C05245=1041.668,269.264,389.932,171.541,41.105,157.842
C05246=1041.675,269.513,389.901,171.543,41.107,157.842
C05247=1041.682,269.761,389.871,171.547,41.109,157.843
C05248=1041.688,270.009,389.840,171.550,41.111,157.843
C05249=1041.695,270.257,389.811,171.553,41.113,157.844
C05250=1041.701,270.505,389.779,171.556,41.115,157.845
C05251=1041.709,270.753,389.749,171.560,41.117,157.845
C05252=1041.714,271.001,389.719,171.562,41.119,157.846
C05253=1041.722,271.249,389.689,171.566,41.121,157.846
C05254=1041.728,271.497,389.657,171.569,41.123,157.847
C05255=1041.735,271.745,389.627,171.572,41.125,157.848
C05256=1041.741,271.993,389.597,171.575,41.127,157.848
C05257=1041.748,272.241,389.565,171.579,41.129,157.849
C05258=1041.755,272.489,389.535,171.581,41.131,157.849
C05259=1041.762,272.738,389.504,171.585,41.133,157.850
C05260=1041.768,272.985,389.473,171.588,41.135,157.851
C05261=1041.775,273.233,389.443,171.591,41.136,157.851
C05262=1041.781,273.482,389.413,171.594,41.139,157.852
C05263=1041.788,273.729,389.381,171.598,41.141,157.853
C05264=1041.795,273.977,389.351,171.600,41.143,157.853
C05265=1041.801,274.225,389.320,171.604,41.145,157.854
C05266=1041.808,274.473,389.289,171.607,41.147,157.854
C05267=1041.815,274.721,389.258,171.610,41.149,157.855
C05268=1041.822,274.970,389.228,171.613,41.151,157.856
C05269=1041.828,275.217,389.196,171.617,41.153,157.856
C05270=1041.835,275.465,389.166,171.619,41.155,157.857
C05271=1041.842,275.713,389.135,171.623,41.157,157.857
C05272=1041.848,275.961,389.104,171.626,41.159,157.858
C05273=1041.855,276.209,389.073,171.630,41.161,157.859
C05274=1041.862,276.457,389.043,171.632,41.163,157.859
C05275=1041.870,276.760,389.005,171.637,41.165,157.860
C05276=1041.878,277.061,388.967,171.641,41.168,157.861
C05277=1041.886,277.364,388.929,171.645,41.171,157.862
C05278=1041.894,277.666,388.891,171.649,41.173,157.862
C05279=1041.900,277.915,388.860,171.651,41.175,157.863
C05280=1041.908,278.162,388.830,171.655,41.177,157.864
C05281=1041.915,278.410,388.798,171.659,41.179,157.864
C05282=1041.921,278.659,388.767,171.661,41.181,157.865
C05283=1041.928,278.906,388.736,171.665,41.183,157.865
C05284=1041.934,279.154,388.705,171.668,41.185,157.866
C05285=1041.941,279.402,388.674,171.671,41.188,157.867
C05286=1041.947,279.650,388.643,171.675,41.190,157.867
C05287=1041.954,279.898,388.611,171.678,41.192,157.868
C05288=1041.960,280.146,388.580,171.682,41.194,157.869
C05289=1041.967,280.394,388.549,171.684,41.196,157.869
C05290=1041.974,280.642,388.517,171.688,41.198,157.870
C05291=1041.981,280.890,388.486,171.691,41.200,157.871
C05292=1041.987,281.138,388.455,171.694,41.202,157.871
C05293=1041.994,281.386,388.424,171.698,41.204,157.872
C05294=1042.001,281.634,388.392,171.701,41.206,157.872
C05295=1042.007,281.882,388.361,171.705,41.208,157.873
C05296=1042.014,282.130,388.329,171.708,41.211,157.874
C05297=1042.021,282.378,388.298,171.711,41.213,157.874
C05298=1042.027,282.626,388.266,171.715,41.215,157.875
C05299=1042.034,282.873,388.235,171.717,41.217,157.876
C05300=1042.041,283.121,388.204,171.721,41.219,157.876
C05301=1042.048,283.369,388.172,171.725,41.221,157.877
C05302=1042.054,283.617,388.141,171.728,41.223,157.878
C05303=1042.061,283.865,388.109,171.732,41.226,157.878
C05304=1042.068,284.113,388.078,171.735,41.228,157.879
C05305=1042.075,284.361,388.046,171.738,41.230,157.880
C05306=1042.081,284.609,388.015,171.742,41.232,157.880
C05307=1042.088,284.857,387.983,171.745,41.234,157.881
C05308=1042.095,285.105,387.952,171.748,41.236,157.882
C05309=1042.101,285.352,387.921,171.752,41.238,157.882
C05310=1042.108,285.600,387.888,171.756,41.240,157.883
C05311=1042.115,285.848,387.857,171.758,41.243,157.884
C05312=1042.122,286.096,387.826,171.762,41.245,157.884
C05313=1042.129,286.343,387.794,171.766,41.247,157.885
C05314=1042.135,286.591,387.763,171.769,41.249,157.886
C05315=1042.142,286.839,387.731,171.772,41.251,157.886
C05316=1042.149,287.087,387.699,171.776,41.253,157.887
C05317=1042.156,287.334,387.668,171.780,41.255,157.888
C05318=1042.162,287.583,387.635,171.782,41.258,157.888
C05319=1042.169,287.831,387.604,171.786,41.260,157.889
C05320=1042.176,288.079,387.572,171.790,41.262,157.890
C05321=1042.183,288.326,387.540,171.793,41.264,157.890
C05322=1042.189,288.575,387.508,171.797,41.267,157.891
C05323=1042.196,288.822,387.476,171.800,41.269,157.892
C05324=1042.203,289.070,387.445,171.804,41.271,157.892
C05325=1042.209,289.318,387.413,171.807,41.273,157.893
C05326=1042.217,289.566,387.381,171.811,41.275,157.894
C05327=1042.223,289.814,387.349,171.814,41.277,157.894
C05328=1042.230,290.061,387.317,171.818,41.279,157.895
C05329=1042.237,290.309,387.285,171.821,41.282,157.896
C05330=1042.243,290.557,387.252,171.825,41.284,157.896
C05331=1042.252,290.871,387.212,171.830,41.287,157.897
C05332=1042.260,291.185,387.171,171.834,41.290,157.898
C05333=1042.269,291.500,387.131,171.839,41.292,157.899
C05334=1042.277,291.813,387.090,171.842,41.295,157.900
C05335=1042.285,292.061,387.058,171.846,41.298,157.901
C05336=1042.291,292.309,387.026,171.850,41.300,157.901
C05337=1042.298,292.557,386.994,171.853,41.302,157.902
C05338=1042.304,292.805,386.962,171.857,41.305,157.903
C05339=1042.311,293.052,386.930,171.860,41.307,157.903
C05340=1042.318,293.300,386.897,171.864,41.309,157.904
C05341=1042.325,293.548,386.866,171.867,41.311,157.905
C05342=1042.331,293.796,386.833,171.871,41.313,157.905
C05343=1042.338,294.043,386.801,171.875,41.315,157.906
C05344=1042.346,294.291,386.769,171.878,41.318,157.907
C05345=1042.352,294.539,386.736,171.882,41.320,157.908
C05346=1042.359,294.786,386.704,171.885,41.323,157.908
C05347=1042.366,295.035,386.672,171.889,41.325,157.909
C05348=1042.373,295.283,386.639,171.893,41.327,157.910
C05349=1042.379,295.530,386.607,171.896,41.330,157.910
C05350=1042.386,295.777,386.575,171.900,41.332,157.911
C05351=1042.393,296.026,386.541,171.904,41.334,157.912
C05352=1042.399,296.273,386.509,171.907,41.336,157.913
C05353=1042.405,296.521,386.476,171.911,41.339,157.913
C05354=1042.412,296.768,386.443,171.915,41.342,157.914
C05355=1042.419,297.016,386.411,171.918,41.344,157.915
C05356=1042.426,297.264,386.378,171.922,41.346,157.916
C05357=1042.432,297.512,386.346,171.925,41.348,157.916
C05358=1042.438,297.760,386.313,171.929,41.351,157.917
C05359=1042.446,298.007,386.280,171.933,41.353,157.918
C05360=1042.452,298.255,386.247,171.937,41.356,157.919
C05361=1042.458,298.502,386.214,171.940,41.358,157.919
C05362=1042.465,298.751,386.181,171.944,41.360,157.920
C05363=1042.472,298.998,386.149,171.947,41.363,157.921
C05364=1042.479,299.246,386.116,171.951,41.365,157.921
C05365=1042.486,299.494,386.083,171.955,41.368,157.922
C05366=1042.492,299.741,386.051,171.959,41.370,157.923
C05367=1042.498,299.989,386.018,171.962,41.372,157.924
C05368=1042.505,300.237,385.985,171.966,41.375,157.924
C05369=1042.512,300.485,385.953,171.970,41.377,157.925
C05370=1042.519,300.732,385.919,171.973,41.380,157.926
C05371=1042.526,300.980,385.886,171.977,41.382,157.927
C05372=1042.532,301.227,385.853,171.981,41.385,157.928
C05373=1042.539,301.476,385.820,171.984,41.387,157.928
C05374=1042.546,301.723,385.788,171.988,41.389,157.929
C05375=1042.553,301.971,385.754,171.992,41.392,157.930
C05376=1042.559,302.218,385.721,171.996,41.394,157.930
C05377=1042.566,302.466,385.689,172.000,41.397,157.931
C05378=1042.573,302.714,385.655,172.004,41.399,157.932
C05379=1042.580,302.961,385.623,172.008,41.401,157.933
C05380=1042.587,303.209,385.590,172.012,41.404,157.934
C05381=1042.593,303.456,385.556,172.014,41.407,157.934
C05382=1042.600,303.704,385.523,172.018,41.409,157.935
C05383=1042.606,303.952,385.490,172.022,41.411,157.936
C05384=1042.614,304.200,385.457,172.026,41.414,157.937
C05385=1042.621,304.447,385.424,172.030,41.417,157.937
C05386=1042.628,304.695,385.391,172.034,41.419,157.938
C05387=1042.637,305.026,385.347,172.039,41.422,157.939
C05388=1042.646,305.356,385.302,172.044,41.425,157.940
C05389=1042.655,305.687,385.258,172.049,41.428,157.941
C05390=1042.664,306.017,385.213,172.054,41.432,157.942
C05391=1042.671,306.265,385.180,172.058,41.435,157.943
C05392=1042.678,306.512,385.147,172.062,41.437,157.944
C05393=1042.685,306.760,385.114,172.066,41.439,157.945
C05394=1042.692,307.007,385.081,172.070,41.442,157.945
C05395=1042.699,307.255,385.047,172.074,41.444,157.946
C05396=1042.706,307.503,385.014,172.078,41.447,157.947
C05397=1042.713,307.750,384.981,172.082,41.449,157.948
C05398=1042.720,307.999,384.947,172.085,41.452,157.948
C05399=1042.726,308.246,384.914,172.089,41.454,157.949
C05400=1042.734,308.493,384.881,172.093,41.457,157.950
C05401=1042.741,308.741,384.848,172.097,41.459,157.951
C05402=1042.748,308.989,384.814,172.101,41.462,157.952
C05403=1042.755,309.236,384.780,172.105,41.464,157.952
C05404=1042.762,309.484,384.747,172.109,41.467,157.953
C05405=1042.769,309.732,384.713,172.114,41.469,157.954
C05406=1042.775,309.979,384.680,172.118,41.472,157.955
C05407=1042.783,310.227,384.646,172.122,41.474,157.956
C05408=1042.790,310.474,384.614,172.126,41.477,157.956
C05409=1042.798,310.722,384.580,172.129,41.479,157.957
C05410=1042.804,310.969,384.546,172.133,41.482,157.958
C05411=1042.811,311.217,384.513,172.137,41.484,157.959
C05412=1042.819,311.464,384.479,172.141,41.487,157.960
C05413=1042.825,311.713,384.446,172.145,41.489,157.960
C05414=1042.833,311.960,384.412,172.149,41.492,157.961
C05415=1042.839,312.207,384.378,172.153,41.494,157.962
C05416=1042.846,312.455,384.344,172.158,41.497,157.963
C05417=1042.854,312.703,384.311,172.162,41.499,157.964
C05418=1042.860,312.951,384.276,172.166,41.503,157.965
C05419=1042.867,313.198,384.243,172.170,41.505,157.965
C05420=1042.873,313.446,384.208,172.174,41.508,157.966
C05421=1042.880,313.693,384.175,172.178,41.510,157.967
C05422=1042.886,313.940,384.140,172.181,41.513,157.968
C05423=1042.894,314.188,384.106,172.186,41.516,157.969
C05424=1042.900,314.436,384.072,172.190,41.519,157.970
C05425=1042.907,314.683,384.038,172.193,41.521,157.970
C05426=1042.915,314.931,384.004,172.197,41.524,157.971
C05427=1042.921,315.178,383.969,172.202,41.527,157.972
C05428=1042.928,315.425,383.935,172.205,41.530,157.973
C05429=1042.934,315.673,383.901,172.210,41.532,157.974
C05430=1042.942,315.921,383.867,172.214,41.535,157.975
C05431=1042.948,316.168,383.832,172.218,41.538,157.976
C05432=1042.955,316.415,383.798,172.222,41.540,157.976
C05433=1042.961,316.663,383.764,172.226,41.543,157.977
C05434=1042.969,316.911,383.730,172.230,41.546,157.978
C05435=1042.975,317.158,383.695,172.234,41.549,157.979
C05436=1042.983,317.406,383.661,172.238,41.551,157.980
C05437=1042.989,317.653,383.626,172.243,41.554,157.981
C05438=1042.997,317.901,383.592,172.247,41.557,157.982
C05439=1043.003,318.149,383.558,172.251,41.560,157.982
C05440=1043.011,318.396,383.523,172.255,41.563,157.983
C05441=1043.016,318.643,383.489,172.259,41.565,157.984
C05442=1043.024,318.890,383.455,172.263,41.568,157.985
C05443=1043.033,319.226,383.408,172.270,41.572,157.986
C05444=1043.042,319.561,383.361,172.275,41.576,157.988
C05445=1043.052,319.896,383.315,172.280,41.579,157.989
C05446=1043.062,320.232,383.267,172.287,41.583,157.990
C05447=1043.069,320.479,383.234,172.291,41.586,157.991
C05448=1043.076,320.727,383.198,172.295,41.589,157.992
C05449=1043.082,320.975,383.164,172.299,41.592,157.993
C05450=1043.090,321.222,383.129,172.304,41.595,157.994
C05451=1043.096,321.469,383.094,172.308,41.597,157.994
C05452=1043.104,321.717,383.061,172.312,41.600,157.995
C05453=1043.110,321.964,383.025,172.316,41.603,157.996
C05454=1043.118,322.211,382.991,172.321,41.606,157.997
C05455=1043.124,322.459,382.956,172.325,41.608,157.998
C05456=1043.132,322.706,382.922,172.329,41.612,157.999
C05457=1043.139,322.954,382.886,172.333,41.614,158.000
